// TwinCAT 3 PLC project PLC
// Title: TcError
// Company: Roald87
// Author: Roald Ruiter
// ProjectVersion: 0.2.2.0
// Description: Translate TwinCAT error codes
// ProgramVersion: 3.1.4023.0
// libraries:
//   Tc2_Standard, * (Beckhoff Automation GmbH)
//   Tc2_System, * (Beckhoff Automation GmbH)
//   Tc3_Module, * (Beckhoff Automation GmbH)
//   TcUnit,1.2.0.0,www.tcunit.org
// project tree:
//   ADS/ AdsErrorCodeDescription.TcPOU, AdsErrorCodes.TcDUT, ToAdsErrorCode.TcPOU
//   NC/ NcErrorCodes.TcDUT, ToNcErrorCode.TcPOU, NcErrorCodeDescription.TcPOU
//   NC_Tests/ ToNcErrorCode_Tests.TcPOU, NcErrorCodeDesciption_Tests.TcPOU
//   / PlcTask.TcTTO, UnitTests.TcPOU
//   Win32/ ToWin32ErrorCode.TcPOU, Win32ErrorCodeDescription.TcPOU, Win32ErrorCodes.TcDUT
//   Win32_Tests/ ToWin32ErrorCode_Tests.TcPOU, Win32ErrorCodeDesciption_Tests.TcPOU
// real-time tasks:
//   TASK PlcTask: cycle T#10ms, priority 20, ADS port 350

CONFIGURATION PLC
    RESOURCE PLC ON TwinCAT3
        TASK PlcTask(INTERVAL := T#10ms, PRIORITY := 20);
        PROGRAM UnitTests WITH PlcTask : UnitTests;
    END_RESOURCE
END_CONFIGURATION

// ---- ADS/AdsErrorCodes.TcDUT
{attribute 'qualified_only'}
{attribute 'strict'}
{attribute 'to_string'}
(*
All ADS error codes.

## Source
https://infosys.beckhoff.com/english.php?content=../content/1033/tf6701_tc3_iot_communication_mqtt/374277003.html&id=
*)
TYPE AdsErrorCodes : (
    ERR_NOERROR := 0,
    ERR_INTERNAL,
    ERR_NORTIME,
    ERR_ALLOCLOCKEDMEM,
    ERR_INSERTMAILBOX,
    ERR_WRONGRECEIVEHMSG,
    ERR_TARGETPORTNOTFOUND,
    ERR_TARGETMACHINENOTFOUND,
    ERR_UNKNOWNCMDID,
    ERR_BADTASKID,
    ERR_NOIO,
    ERR_UNKNOWNAMSCMD,
    ERR_WIN32ERROR,
    ERR_PORTNOTCONNECTED,
    ERR_INVALIDAMSLENGTH,
    ERR_INVALIDAMSNETID,
    ERR_LOWINSTLEVEL,
    ERR_NODEBUGINTAVAILABLE,
    ERR_PORTDISABLED,
    ERR_PORTALREADYCONNECTED,
    ERR_AMSSYNC_W32ERROR,
    ERR_AMSSYNC_TIMEOUT,
    ERR_AMSSYNC_AMSERROR,
    ERR_AMSSYNC_NOINDEXINMAP,
    ERR_INVALIDAMSPORT,
    ERR_NOMEMORY,
    ERR_TCPSEND,
    ERR_HOSTUNREACHABLE,
    ERR_INVALIDAMSFRAGMENT,
    ERR_TLSSEND,
    ERR_ACCESSDENIED,
    ROUTERERR_NOLOCKEDMEMORY := 1280,
    ROUTERERR_RESIZEMEMORY := 1281,
    ROUTERERR_MAILBOXFULL := 1282,
    ROUTERERR_DEBUGBOXFULL := 1283,
    ROUTERERR_UNKNOWNPORTTYPE := 1284,
    ROUTERERR_NOTINITIALIZED := 1285,
    ROUTERERR_PORTALREADYINUSE := 1286,
    ROUTERERR_NOTREGISTERED := 1287,
    ROUTERERR_NOMOREQUEUES := 1288,
    ROUTERERR_INVALIDPORT := 1289,
    ROUTERERR_NOTACTIVATED := 1290,
    ROUTERERR_FRAGMENTBOXFULL := 1291,
    ROUTERERR_FRAGMENTTIMEOUT := 1292,
    ROUTERERR_TOBEREMOVED := 1293,
    ADSERR_DEVICE_ERROR := 1792,
    ADSERR_DEVICE_SRVNOTSUPP := 1793,
    ADSERR_DEVICE_INVALIDGRP := 1794,
    ADSERR_DEVICE_INVALIDOFFSET := 1795,
    ADSERR_DEVICE_INVALIDACCESS := 1796,
    ADSERR_DEVICE_INVALIDSIZE := 1797,
    ADSERR_DEVICE_INVALIDDATA := 1798,
    ADSERR_DEVICE_NOTREADY := 1799,
    ADSERR_DEVICE_BUSY := 1800,
    ADSERR_DEVICE_INVALIDCONTEXT := 1801,
    ADSERR_DEVICE_NOMEMORY := 1802,
    ADSERR_DEVICE_INVALIDPARM := 1803,
    ADSERR_DEVICE_NOTFOUND := 1804,
    ADSERR_DEVICE_SYNTAX := 1805,
    ADSERR_DEVICE_INCOMPATIBLE := 1806,
    ADSERR_DEVICE_EXISTS := 1807,
    ADSERR_DEVICE_SYMBOLNOTFOUND := 1808,
    ADSERR_DEVICE_SYMBOLVERSIONINVALID := 1809,
    ADSERR_DEVICE_INVALIDSTATE := 1810,
    ADSERR_DEVICE_TRANSMODENOTSUPP := 1811,
    ADSERR_DEVICE_NOTIFYHNDINVALID := 1812,
    ADSERR_DEVICE_CLIENTUNKNOWN := 1813,
    ADSERR_DEVICE_NOMOREHDLS := 1814,
    ADSERR_DEVICE_INVALIDWATCHSIZE := 1815,
    ADSERR_DEVICE_NOTINIT := 1816,
    ADSERR_DEVICE_TIMEOUT := 1817,
    ADSERR_DEVICE_NOINTERFACE := 1818,
    ADSERR_DEVICE_INVALIDINTERFACE := 1819,
    ADSERR_DEVICE_INVALIDCLSID := 1820,
    ADSERR_DEVICE_INVALIDOBJID := 1821,
    ADSERR_DEVICE_PENDING := 1822,
    ADSERR_DEVICE_ABORTED := 1823,
    ADSERR_DEVICE_WARNING := 1824,
    ADSERR_DEVICE_INVALIDARRAYIDX := 1825,
    ADSERR_DEVICE_SYMBOLNOTACTIVE := 1826,
    ADSERR_DEVICE_ACCESSDENIED := 1827,
    ADSERR_DEVICE_LICENSENOTFOUND := 1828,
    ADSERR_DEVICE_LICENSEEXPIRED := 1829,
    ADSERR_DEVICE_LICENSEEXCEEDED := 1830,
    ADSERR_DEVICE_LICENSEINVALID := 1831,
    ADSERR_DEVICE_LICENSESYSTEMID := 1832,
    ADSERR_DEVICE_LICENSENOTIMELIMIT := 1833,
    ADSERR_DEVICE_LICENSEFUTUREISSUE := 1834,
    ADSERR_DEVICE_LICENSETIMETOLONG := 1835,
    ADSERR_DEVICE_EXCEPTION := 1836,
    ADSERR_DEVICE_LICENSEDUPLICATED := 1837,
    ADSERR_DEVICE_SIGNATUREINVALID := 1838,
    ADSERR_DEVICE_CERTIFICATEINVALID := 1839,
    ADSERR_DEVICE_LICENSEOEMNOTFOUND := 1840,
    ADSERR_DEVICE_LICENSERESTRICTED := 1841,
    ADSERR_DEVICE_LICENSEDEMODENIED := 1842,
    ADSERR_DEVICE_INVALIDFNCID := 1843,
    ADSERR_DEVICE_OUTOFRANGE := 1844,
    ADSERR_DEVICE_INVALIDALIGNMENT := 1845,
    ADSERR_DEVICE_LICENSEPLATFORM := 1846,
    ADSERR_DEVICE_FORWARD_PL := 1847,
    ADSERR_DEVICE_FORWARD_DL := 1848,
    ADSERR_DEVICE_FORWARD_RT := 1849,
    ADSERR_CLIENT_ERROR := 1856,
    ADSERR_CLIENT_INVALIDPARM := 1857,
    ADSERR_CLIENT_LISTEMPTY := 1858,
    ADSERR_CLIENT_VARUSED := 1859,
    ADSERR_CLIENT_DUPLINVOKEID := 1860,
    ADSERR_CLIENT_SYNCTIMEOUT := 1861,
    ADSERR_CLIENT_W32ERROR := 1862,
    ADSERR_CLIENT_TIMEOUTINVALID := 1863,
    ADSERR_CLIENT_PORTNOTOPEN := 1864,
    ADSERR_CLIENT_NOAMSADDR := 1865,
    ADSERR_CLIENT_SYNCINTERNAL := 1872,
    ADSERR_CLIENT_ADDHASH := 1873,
    ADSERR_CLIENT_REMOVEHASH := 1874,
    ADSERR_CLIENT_NOMORESYM := 1875,
    ADSERR_CLIENT_SYNCRESINVALID := 1876,
    ADSERR_CLIENT_SYNCPORTLOCKED := 1877,
    RTERR_INTERNAL := 4096,
    RTERR_BADTIMERPERIODS := 4097,
    RTERR_INVALIDTASKPTR := 4098,
    RTERR_INVALIDSTACKPTR := 4099,
    RTERR_PRIOEXISTS := 4100,
    RTERR_NOMORETCB := 4101,
    RTERR_NOMORESEMAS := 4102,
    RTERR_NOMOREQUEUES := 4103,
    RTERR_EXTIRQALREADYDEF := 4109,
    RTERR_EXTIRQNOTDEF := 4110,
    RTERR_EXTIRQINSTALLFAILED := 4111,
    RTERR_IRQLNOTLESSOREQUAL := 4112,
    RTERR_VMXNOTSUPPORTED := 4119,
    RTERR_VMXDISABLED := 4120,
    RTERR_VMXCONTROLSMISSING := 4121,
    RTERR_VMXENABLEFAILS := 4122,
    WSAETIMEDOUT := 10060,
    WSAECONNREFUSED := 10061,
    WSAEHOSTUNREACH := 10065,
    ERR_UNKNOWN := 4294967294
) UDINT;
END_TYPE

// ---- NC/NcErrorCodes.TcDUT
{attribute 'qualified_only'}
{attribute 'strict'}
(*
Some NC Error codes

Source: https://infosys.beckhoff.com/content/1033/tc3ncerrcode/1521556875.html?id=2911757239699425890
*)
TYPE NcErrorCodes : (
    NO_ERROR := 0,
    CONTROLLER_ERROR_CONTROLLER_ID_NOT_ALLOWED := 17664,
    CONTROLLER_ERROR_CONTROLLER_TYPE_NOT_ALLOWED := 17665,
    CONTROLLER_ERROR_OPERATION_MODE_CONTROLLER_NOT_ALLOWED := 17666,
    CONTROLLER_ERROR_WEIGHTING_OF_THE_VELOCITY_PRE_CONTROL_NOT_ALLOWED := 17667,
    CONTROLLER_ERROR_LAG_ERROR_MONITOR_POSITION_NOT_ALLOWED := 17668,
    CONTROLLER_ERROR_LAG_MONITORING_VELOCITY_NOT_ALLOWED := 17669,
    CONTROLLER_ERROR_LAG_ERROR_WINDOW_POSITION_NOT_ALLOWED := 17670,
    CONTROLLER_ERROR_LAG_ERROR_FILTER_TIME_POSITION_NOT_ALLOWED := 17671,
    CONTROLLER_ERROR_LAG_ERROR_WINDOW_VELOCITY_NOT_ALLOWED := 17672,
    CONTROLLER_ERROR_LAG_ERROR_FILTER_TIME_VELOCITY_NOT_ALLOWED := 17673,
    CONTROLLER_ERROR_CONTROLLER_OUTPUT_LIMITATION_OUTPUT_LIMITATION_NOT_ALLOWED := 17674,
    CONTROLLER_ERROR_PROPORTIONAL_GAIN_KV_OR_KP_CONTROLLER_NOT_ALLOWED := 17680,
    CONTROLLER_ERROR_INTEGRAL_ACTION_TIME_TN_CONTROLLER_NOT_ALLOWED_POSITION := 17681,
    CONTROLLER_ERROR_RATE_TIME_TV_CONTROLLER_NOT_ALLOWED_POSITION := 17682,
    CONTROLLER_ERROR_DAMPING_TIME_TD_CONTROLLER_NOT_ALLOWED_POSITION := 17683,
    CONTROLLER_ERROR_ACTIVATION_OF_THE_AUTOMATIC_OFFSET_CALIBRATION_NOT_ALLOWED := 17684,
    CONTROLLER_ERROR_ADDITIONAL_PROPORTIONAL_GAIN_KV_OR_KP_CONTROLLER_NOT_ALLOWED := 17685,
    CONTROLLER_ERROR_REFERENCE_VELOCITY_FOR_ADDITIONAL_PROP_GAIN_CONTROLLER_NOT_ALLOWED := 17686,
    CONTROLLER_ERROR_PROPORTIONAL_GAIN_PA_PROPORTION_NOT_ALLOWED := 17687,
    CONTROLLER_ERROR_PROPORTIONAL_GAIN_KV_CONTROLLER_NOT_ALLOWED := 17688,
    CONTROLLER_ERROR_INTEGRAL_ACTION_TIME_TN_CONTROLLER_NOT_ALLOWED_VELOCITY := 17689,
    CONTROLLER_ERROR_VELOCITY_FILTER_TIME_NOT_ALLOWED := 17692,
    CONTROLLER_ERROR_DEAD_RANGE_NOT_ALLOWED := 17693,
    CONTROLLER_ERROR_PROPORTIONAL_GAIN_KCP_NOT_ALLOWED := 17695,
    CONTROLLER_ERROR_RATE_TIME_TV_CONTROLLER_NOT_ALLOWED := 17696,
    CONTROLLER_ERROR_DAMPING_TIME_TD_CONTROLLER_NOT_ALLOWED := 17697,
    CONTROLLER_ERROR_LIMITATION_OF_THE_I_PART_NOT_ALLOWED := 17698,
    CONTROLLER_ERROR_LIMITATION_OF_THE_D_PART_NOT_ALLOWED := 17699,
    CONTROLLER_ERROR_PARAMETER_DEACTIVATION_OF_THE_I_PART_DURING_TRAVEL_NOT_ALLOWED := 17700,
    CONTROLLER_ERROR_PARAMETER_FILTER_TIME_FOR_P_T2_FILTER_NOT_ALLOWED := 17701,
    CONTROLLER_ERROR_VELOCITY_OBSERVER_PARAMETERIZED_MODE_IS_NOT_ALLOWED := 17702,
    CONTROLLER_ERROR_VELOCITY_OBSERVER_MOTOR_TORQUE_CONSTANT_KT_OR_KF_IS_NOT_ALLOWED := 17703,
    CONTROLLER_ERROR_VELOCITY_OBSERVER_MOTOR_MOMENT_OF_INERTIA_JM_IS_NOT_ALLOWED := 17704,
    CONTROLLER_ERROR_VELOCITY_OBSERVER_BANDWIDTH_F0_IS_NOT_ALLOWED := 17705,
    CONTROLLER_ERROR_VELOCITY_OBSERVER_CORRECTION_FACTOR_KC_IS_NOT_ALLOWED := 17706,
    CONTROLLER_ERROR_VELOCITY_OBSERVER_TIME_CONSTANT_T_FOR_1ST_ORDER_FILTER_NOT_ALLOWED := 17707,
    CONTROLLER_ERROR_VELOCITY_OBSERVER_AMPLITUDE_DAMPING_FOR_2ND_ORDER_FILTER_NOT_ALLOWED := 17708,
    CONTROLLER_ERROR_VELOCITY_OBSERVER_FREQUENCY_FOR_2ND_ORDER_FILTER_NOT_ALLOWED := 17709,
    CONTROLLER_ERROR_CONTROLLER_INITIALIZATION := 17728,
    CONTROLLER_ERROR_AXIS_ADDRESS := 17729,
    CONTROLLER_ERROR_DRIVE_ADDRESS := 17730,
    CONTROLLER_ERROR_LAG_ERROR_MONITOR_POSITION := 17744,
    CONTROLLER_ERROR_LAG_MONITORING_VELOCITY := 17745,
    CONTROLLER_ERROR_INTERNAL_ERROR_CONTROLERR_RANGE_AREA_ASIDE := 17824,
    CONTROLLER_ERROR_INTERNAL_ERROR_CONTROLERR_RANGE_AREA_BSIDE := 17825,
    CONTROLLER_ERROR_INTERNAL_ERROR_CONTROLERR_RANGE_QNENN := 17826,
    CONTROLLER_ERROR_INTERNAL_ERROR_CONTROLERR_RANGE_PNENN := 17827,
    CONTROLLER_ERROR_INTERNAL_ERROR_CONTROLERR_RANGE_AXISIDPRESP0 := 17828,
    ERR_UNKNOWN := 65535
);
END_TYPE

// ---- Win32/Win32ErrorCodes.TcDUT
{attribute 'qualified_only'}
{attribute 'strict'}
{attribute 'to_string'}
(*
All Win32 error codes.

## Source
https://infosys.beckhoff.com/content/1033/devicemanager/391166347.html?id=8711134805786442486
*)
TYPE Win32ErrorCodes : (
    ERROR_SUCCESS := 0,
    ERROR_INVALID_FUNCTION := 1,
    ERROR_FILE_NOT_FOUND := 2,
    ERROR_PATH_NOT_FOUND := 3,
    ERROR_TOO_MANY_OPEN_FILES := 4,
    ERROR_ACCESS_DENIED := 5,
    ERROR_INVALID_HANDLE := 6,
    ERROR_ARENA_TRASHED := 7,
    ERROR_NOT_ENOUGH_MEMORY := 8,
    ERROR_INVALID_BLOCK := 9,
    ERROR_BAD_ENVIRONMENT := 10,
    ERROR_BAD_FORMAT := 11,
    ERROR_INVALID_ACCESS := 12,
    ERROR_INVALID_DATA := 13,
    ERROR_OUTOFMEMORY := 14,
    ERROR_INVALID_DRIVE := 15,
    ERROR_CURRENT_DIRECTORY := 16,
    ERROR_NOT_SAME_DEVICE := 17,
    ERROR_NO_MORE_FILES := 18,
    ERROR_WRITE_PROTECT := 19,
    ERROR_BAD_UNIT := 20,
    ERROR_NOT_READY := 21,
    ERROR_BAD_COMMAND := 22,
    ERROR_CRC := 23,
    ERROR_BAD_LENGTH := 24,
    ERROR_SEEK := 25,
    ERROR_NOT_DOS_DISK := 26,
    ERROR_SECTOR_NOT_FOUND := 27,
    ERROR_OUT_OF_PAPER := 28,
    ERROR_WRITE_FAULT := 29,
    ERROR_READ_FAULT := 30,
    ERROR_GEN_FAILURE := 31,
    ERROR_SHARING_VIOLATION := 32,
    ERROR_LOCK_VIOLATION := 33,
    ERROR_WRONG_DISK := 34,
    ERROR_SHARING_BUFFER_EXCEEDED := 36,
    ERROR_HANDLE_EOF := 38,
    ERROR_HANDLE_DISK_FULL := 39,
    ERROR_NOT_SUPPORTED := 50,
    ERROR_REM_NOT_LIST := 51,
    ERROR_DUP_NAME := 52,
    ERROR_BAD_NETPATH := 53,
    ERROR_NETWORK_BUSY := 54,
    ERROR_DEV_NOT_EXIST := 55,
    ERROR_TOO_MANY_CMDS := 56,
    ERROR_ADAP_HDW_ERR := 57,
    ERROR_BAD_NET_RESP := 58,
    ERROR_UNEXP_NET_ERR := 59,
    ERROR_BAD_REM_ADAP := 60,
    ERROR_PRINTQ_FULL := 61,
    ERROR_NO_SPOOL_SPACE := 62,
    ERROR_PRINT_CANCELLED := 63,
    ERROR_NETNAME_DELETED := 64,
    ERROR_NETWORK_ACCESS_DENIED := 65,
    ERROR_BAD_DEV_TYPE := 66,
    ERROR_BAD_NET_NAME := 67,
    ERROR_TOO_MANY_NAMES := 68,
    ERROR_TOO_MANY_SESS := 69,
    ERROR_SHARING_PAUSED := 70,
    ERROR_REQ_NOT_ACCEP := 71,
    ERROR_REDIR_PAUSED := 72,
    ERROR_FILE_EXISTS := 80,
    ERROR_CANNOT_MAKE := 82,
    ERROR_FAIL_I24 := 83,
    ERROR_OUT_OF_STRUCTURES := 84,
    ERROR_ALREADY_ASSIGNED := 85,
    ERROR_INVALID_PASSWORD := 86,
    ERROR_INVALID_PARAMETER := 87,
    ERROR_NET_WRITE_FAULT := 88,
    ERROR_NO_PROC_SLOTS := 89,
    ERROR_TOO_MANY_SEMAPHORES := 100,
    ERROR_EXCL_SEM_ALREADY_OWNED := 101,
    ERROR_SEM_IS_SET := 102,
    ERROR_TOO_MANY_SEM_REQUESTS := 103,
    ERROR_INVALID_AT_INTERRUPT_TIME := 104,
    ERROR_SEM_OWNER_DIED := 105,
    ERROR_SEM_USER_LIMIT := 106,
    ERROR_DISK_CHANGE := 107,
    ERROR_DRIVE_LOCKED := 108,
    ERROR_BROKEN_PIPE := 109,
    ERROR_OPEN_FAILED := 110,
    ERROR_BUFFER_OVERFLOW := 111,
    ERROR_DISK_FULL := 112,
    ERROR_NO_MORE_SEARCH_HANDLES := 113,
    ERROR_INVALID_TARGET_HANDLE := 114,
    ERROR_INVALID_CATEGORY := 117,
    ERROR_INVALID_VERIFY_SWITCH := 118,
    ERROR_BAD_DRIVER_LEVEL := 119,
    ERROR_CALL_NOT_IMPLEMENTED := 120,
    ERROR_SEM_TIMEOUT := 121,
    ERROR_INSUFFICIENT_BUFFER := 122,
    ERROR_INVALID_NAME := 123,
    ERROR_INVALID_LEVEL := 124,
    ERROR_NO_VOLUME_LABEL := 125,
    ERROR_MOD_NOT_FOUND := 126,
    ERROR_PROC_NOT_FOUND := 127,
    ERROR_WAIT_NO_CHILDREN := 128,
    ERROR_CHILD_NOT_COMPLETE := 129,
    ERROR_DIRECT_ACCESS_HANDLE := 130,
    ERROR_NEGATIVE_SEEK := 131,
    ERROR_SEEK_ON_DEVICE := 132,
    ERROR_IS_JOIN_TARGET := 133,
    ERROR_IS_JOINED := 134,
    ERROR_IS_SUBSTED := 135,
    ERROR_NOT_JOINED := 136,
    ERROR_NOT_SUBSTED := 137,
    ERROR_JOIN_TO_JOIN := 138,
    ERROR_SUBST_TO_SUBST := 139,
    ERROR_JOIN_TO_SUBST := 140,
    ERROR_SUBST_TO_JOIN := 141,
    ERROR_BUSY_DRIVE := 142,
    ERROR_SAME_DRIVE := 143,
    ERROR_DIR_NOT_ROOT := 144,
    ERROR_DIR_NOT_EMPTY := 145,
    ERROR_IS_SUBST_PATH := 146,
    ERROR_IS_JOIN_PATH := 147,
    ERROR_PATH_BUSY := 148,
    ERROR_IS_SUBST_TARGET := 149,
    ERROR_SYSTEM_TRACE := 150,
    ERROR_INVALID_EVENT_COUNT := 151,
    ERROR_TOO_MANY_MUXWAITERS := 152,
    ERROR_INVALID_LIST_FORMAT := 153,
    ERROR_LABEL_TOO_LONG := 154,
    ERROR_TOO_MANY_TCBS := 155,
    ERROR_SIGNAL_REFUSED := 156,
    ERROR_DISCARDED := 157,
    ERROR_NOT_LOCKED := 158,
    ERROR_BAD_THREADID_ADDR := 159,
    ERROR_BAD_ARGUMENTS := 160,
    ERROR_BAD_PATHNAME := 161,
    ERROR_SIGNAL_PENDING := 162,
    ERROR_MAX_THRDS_REACHED := 164,
    ERROR_LOCK_FAILED := 167,
    ERROR_BUSY := 170,
    ERROR_CANCEL_VIOLATION := 173,
    ERROR_ATOMIC_LOCKS_NOT_SUPPORTED := 174,
    ERROR_INVALID_SEGMENT_NUMBER := 180,
    ERROR_INVALID_ORDINAL := 182,
    ERROR_ALREADY_EXISTS := 183,
    ERROR_INVALID_FLAG_NUMBER := 186,
    ERROR_SEM_NOT_FOUND := 187,
    ERROR_INVALID_STARTING_CODESEG := 188,
    ERROR_INVALID_STACKSEG := 189,
    ERROR_INVALID_MODULETYPE := 190,
    ERROR_INVALID_EXE_SIGNATURE := 191,
    ERROR_EXE_MARKED_INVALID := 192,
    ERROR_BAD_EXE_FORMAT := 193,
    ERROR_ITERATED_DATA_EXCEEDS_64k := 194,
    ERROR_INVALID_MINALLOCSIZE := 195,
    ERROR_DYNLINK_FROM_INVALID_RING := 196,
    ERROR_IOPL_NOT_ENABLED := 197,
    ERROR_INVALID_SEGDPL := 198,
    ERROR_AUTODATASEG_EXCEEDS_64k := 199,
    ERROR_RING2SEG_MUST_BE_MOVABLE := 200,
    ERROR_RELOC_CHAIN_XEEDS_SEGLIM := 201,
    ERROR_INFLOOP_IN_RELOC_CHAIN := 202,
    ERROR_ENVVAR_NOT_FOUND := 203,
    ERROR_NO_SIGNAL_SENT := 205,
    ERROR_FILENAME_EXCED_RANGE := 206,
    ERROR_RING2_STACK_IN_USE := 207,
    ERROR_META_EXPANSION_TOO_LONG := 208,
    ERROR_INVALID_SIGNAL_NUMBER := 209,
    ERROR_THREAD_1_INACTIVE := 210,
    ERROR_LOCKED := 212,
    ERROR_TOO_MANY_MODULES := 214,
    ERROR_NESTING_NOT_ALLOWED := 215,
    ERROR_EXE_MACHINE_TYPE_MISMATCH := 216,
    ERROR_BAD_PIPE := 230,
    ERROR_PIPE_BUSY := 231,
    ERROR_NO_DATA := 232,
    ERROR_PIPE_NOT_CONNECTED := 233,
    ERROR_MORE_DATA := 234,
    ERROR_VC_DISCONNECTED := 240,
    ERROR_INVALID_EA_NAME := 254,
    ERROR_EA_LIST_INCONSISTENT := 255,
    WAIT_TIMEOUT := 258,
    ERROR_NO_MORE_ITEMS := 259,
    ERROR_CANNOT_COPY := 266,
    ERROR_DIRECTORY := 267,
    ERROR_EAS_DIDNT_FIT := 275,
    ERROR_EA_FILE_CORRUPT := 276,
    ERROR_EA_TABLE_FULL := 277,
    ERROR_INVALID_EA_HANDLE := 278,
    ERROR_EAS_NOT_SUPPORTED := 282,
    ERROR_NOT_OWNER := 288,
    ERROR_TOO_MANY_POSTS := 298,
    ERROR_PARTIAL_COPY := 299,
    ERROR_OPLOCK_NOT_GRANTED := 300,
    ERROR_INVALID_OPLOCK_PROTOCOL := 301,
    ERROR_DISK_TOO_FRAGMENTED := 302,
    ERROR_DELETE_PENDING := 303,
    ERROR_MR_MID_NOT_FOUND := 317,
    ERROR_INVALID_ADDRESS := 487,
    ERROR_ARITHMETIC_OVERFLOW := 534,
    ERROR_PIPE_CONNECTED := 535,
    ERROR_PIPE_LISTENING := 536,
    ERROR_EA_ACCESS_DENIED := 994,
    ERROR_OPERATION_ABORTED := 995,
    ERROR_IO_INCOMPLETE := 996,
    ERROR_IO_PENDING := 997,
    ERROR_NOACCESS := 998,
    ERROR_SWAPERROR := 999,
    ERROR_STACK_OVERFLOW := 1001,
    ERROR_INVALID_MESSAGE := 1002,
    ERROR_CAN_NOT_COMPLETE := 1003,
    ERROR_INVALID_FLAGS := 1004,
    ERROR_UNRECOGNIZED_VOLUME := 1005,
    ERROR_FILE_INVALID := 1006,
    ERROR_FULLSCREEN_MODE := 1007,
    ERROR_NO_TOKEN := 1008,
    ERROR_BADDB := 1009,
    ERROR_BADKEY := 1010,
    ERROR_CANTOPEN := 1011,
    ERROR_CANTREAD := 1012,
    ERROR_CANTWRITE := 1013,
    ERROR_REGISTRY_RECOVERED := 1014,
    ERROR_REGISTRY_CORRUPT := 1015,
    ERROR_REGISTRY_IO_FAILED := 1016,
    ERROR_NOT_REGISTRY_FILE := 1017,
    ERROR_KEY_DELETED := 1018,
    ERROR_NO_LOG_SPACE := 1019,
    ERROR_KEY_HAS_CHILDREN := 1020,
    ERROR_CHILD_MUST_BE_VOLATILE := 1021,
    ERROR_NOTIFY_ENUM_DIR := 1022,
    ERROR_DEPENDENT_SERVICES_RUNNING := 1051,
    ERROR_INVALID_SERVICE_CONTROL := 1052,
    ERROR_SERVICE_REQUEST_TIMEOUT := 1053,
    ERROR_SERVICE_NO_THREAD := 1054,
    ERROR_SERVICE_DATABASE_LOCKED := 1055,
    ERROR_SERVICE_ALREADY_RUNNING := 1056,
    ERROR_INVALID_SERVICE_ACCOUNT := 1057,
    ERROR_SERVICE_DISABLED := 1058,
    ERROR_CIRCULAR_DEPENDENCY := 1059,
    ERROR_SERVICE_DOES_NOT_EXIST := 1060,
    ERROR_SERVICE_CANNOT_ACCEPT_CTRL := 1061,
    ERROR_SERVICE_NOT_ACTIVE := 1062,
    ERROR_FAILED_SERVICE_CONTROLLER_CONNECT := 1063,
    ERROR_EXCEPTION_IN_SERVICE := 1064,
    ERROR_DATABASE_DOES_NOT_EXIST := 1065,
    ERROR_SERVICE_SPECIFIC_ERROR := 1066,
    ERROR_PROCESS_ABORTED := 1067,
    ERROR_SERVICE_DEPENDENCY_FAIL := 1068,
    ERROR_SERVICE_LOGON_FAILED := 1069,
    ERROR_SERVICE_START_HANG := 1070,
    ERROR_INVALID_SERVICE_LOCK := 1071,
    ERROR_SERVICE_MARKED_FOR_DELETE := 1072,
    ERROR_SERVICE_EXISTS := 1073,
    ERROR_ALREADY_RUNNING_LKG := 1074,
    ERROR_SERVICE_DEPENDENCY_DELETED := 1075,
    ERROR_BOOT_ALREADY_ACCEPTED := 1076,
    ERROR_SERVICE_NEVER_STARTED := 1077,
    ERROR_DUPLICATE_SERVICE_NAME := 1078,
    ERROR_DIFFERENT_SERVICE_ACCOUNT := 1079,
    ERROR_CANNOT_DETECT_DRIVER_FAILURE := 1080,
    ERROR_CANNOT_DETECT_PROCESS_ABORT := 1081,
    ERROR_NO_RECOVERY_PROGRAM := 1082,
    ERROR_SERVICE_NOT_IN_EXE := 1083,
    ERROR_NOT_SAFEBOOT_SERVICE := 1084,
    ERROR_END_OF_MEDIA := 1100,
    ERROR_FILEMARK_DETECTED := 1101,
    ERROR_BEGINNING_OF_MEDIA := 1102,
    ERROR_SETMARK_DETECTED := 1103,
    ERROR_NO_DATA_DETECTED := 1104,
    ERROR_PARTITION_FAILURE := 1105,
    ERROR_INVALID_BLOCK_LENGTH := 1106,
    ERROR_DEVICE_NOT_PARTITIONED := 1107,
    ERROR_UNABLE_TO_LOCK_MEDIA := 1108,
    ERROR_UNABLE_TO_UNLOAD_MEDIA := 1109,
    ERROR_MEDIA_CHANGED := 1110,
    ERROR_BUS_RESET := 1111,
    ERROR_NO_MEDIA_IN_DRIVE := 1112,
    ERROR_NO_UNICODE_TRANSLATION := 1113,
    ERROR_DLL_INIT_FAILED := 1114,
    ERROR_SHUTDOWN_IN_PROGRESS := 1115,
    ERROR_NO_SHUTDOWN_IN_PROGRESS := 1116,
    ERROR_IO_DEVICE := 1117,
    ERROR_SERIAL_NO_DEVICE := 1118,
    ERROR_IRQ_BUSY := 1119,
    ERROR_MORE_WRITES := 1120,
    ERROR_COUNTER_TIMEOUT := 1121,
    ERROR_FLOPPY_ID_MARK_NOT_FOUND := 1122,
    ERROR_FLOPPY_WRONG_CYLINDER := 1123,
    ERROR_FLOPPY_UNKNOWN_ERROR := 1124,
    ERROR_FLOPPY_BAD_REGISTERS := 1125,
    ERROR_DISK_RECALIBRATE_FAILED := 1126,
    ERROR_DISK_OPERATION_FAILED := 1127,
    ERROR_DISK_RESET_FAILED := 1128,
    ERROR_EOM_OVERFLOW := 1129,
    ERROR_NOT_ENOUGH_SERVER_MEMORY := 1130,
    ERROR_POSSIBLE_DEADLOCK := 1131,
    ERROR_MAPPED_ALIGNMENT := 1132,
    ERROR_SET_POWER_STATE_VETOED := 1140,
    ERROR_SET_POWER_STATE_FAILED := 1141,
    ERROR_TOO_MANY_LINKS := 1142,
    ERROR_OLD_WIN_VERSION := 1150,
    ERROR_APP_WRONG_OS := 1151,
    ERROR_SINGLE_INSTANCE_APP := 1152,
    ERROR_RMODE_APP := 1153,
    ERROR_INVALID_DLL := 1154,
    ERROR_NO_ASSOCIATION := 1155,
    ERROR_DDE_FAIL := 1156,
    ERROR_DLL_NOT_FOUND := 1157,
    ERROR_NO_MORE_USER_HANDLES := 1158,
    ERROR_MESSAGE_SYNC_ONLY := 1159,
    ERROR_SOURCE_ELEMENT_EMPTY := 1160,
    ERROR_DESTINATION_ELEMENT_FULL := 1161,
    ERROR_ILLEGAL_ELEMENT_ADDRESS := 1162,
    ERROR_MAGAZINE_NOT_PRESENT := 1163,
    ERROR_DEVICE_REINITIALIZATION_NEEDED := 1164,
    ERROR_DEVICE_REQUIRES_CLEANING := 1165,
    ERROR_DEVICE_DOOR_OPEN := 1166,
    ERROR_DEVICE_NOT_CONNECTED := 1167,
    ERROR_NOT_FOUND := 1168,
    ERROR_NO_MATCH := 1169,
    ERROR_SET_NOT_FOUND := 1170,
    ERROR_POINT_NOT_FOUND := 1171,
    ERROR_NO_TRACKING_SERVICE := 1172,
    ERROR_NO_VOLUME_ID := 1173,
    ERROR_UNABLE_TO_REMOVE_REPLACED := 1175,
    ERROR_UNABLE_TO_MOVE_REPLACEMENT := 1176,
    ERROR_UNABLE_TO_MOVE_REPLACEMENT_2 := 1177,
    ERROR_JOURNAL_DELETE_IN_PROGRESS := 1178,
    ERROR_JOURNAL_NOT_ACTIVE := 1179,
    ERROR_POTENTIAL_FILE_FOUND := 1180,
    ERROR_JOURNAL_ENTRY_DELETED := 1181,
    ERROR_BAD_DEVICE := 1200,
    ERROR_CONNECTION_UNAVAIL := 1201,
    ERROR_DEVICE_ALREADY_REMEMBERED := 1202,
    ERROR_NO_NET_OR_BAD_PATH := 1203,
    ERROR_BAD_PROVIDER := 1204,
    ERROR_CANNOT_OPEN_PROFILE := 1205,
    ERROR_BAD_PROFILE := 1206,
    ERROR_NOT_CONTAINER := 1207,
    ERROR_EXTENDED_ERROR := 1208,
    ERROR_INVALID_GROUPNAME := 1209,
    ERROR_INVALID_COMPUTERNAME := 1210,
    ERROR_INVALID_EVENTNAME := 1211,
    ERROR_INVALID_DOMAINNAME := 1212,
    ERROR_INVALID_SERVICENAME := 1213,
    ERROR_INVALID_NETNAME := 1214,
    ERROR_INVALID_SHARENAME := 1215,
    ERROR_INVALID_PASSWORDNAME := 1216,
    ERROR_INVALID_MESSAGENAME := 1217,
    ERROR_INVALID_MESSAGEDEST := 1218,
    ERROR_SESSION_CREDENTIAL_CONFLICT := 1219,
    ERROR_REMOTE_SESSION_LIMIT_EXCEEDED := 1220,
    ERROR_DUP_DOMAINNAME := 1221,
    ERROR_NO_NETWORK := 1222,
    ERROR_CANCELLED := 1223,
    ERROR_USER_MAPPED_FILE := 1224,
    ERROR_CONNECTION_REFUSED := 1225,
    ERROR_GRACEFUL_DISCONNECT := 1226,
    ERROR_ADDRESS_ALREADY_ASSOCIATED := 1227,
    ERROR_ADDRESS_NOT_ASSOCIATED := 1228,
    ERROR_CONNECTION_INVALID := 1229,
    ERROR_CONNECTION_ACTIVE := 1230,
    ERROR_NETWORK_UNREACHABLE := 1231,
    ERROR_HOST_UNREACHABLE := 1232,
    ERROR_PROTOCOL_UNREACHABLE := 1233,
    ERROR_PORT_UNREACHABLE := 1234,
    ERROR_REQUEST_ABORTED := 1235,
    ERROR_CONNECTION_ABORTED := 1236,
    ERROR_RETRY := 1237,
    ERROR_CONNECTION_COUNT_LIMIT := 1238,
    ERROR_LOGIN_TIME_RESTRICTION := 1239,
    ERROR_LOGIN_WKSTA_RESTRICTION := 1240,
    ERROR_INCORRECT_ADDRESS := 1241,
    ERROR_ALREADY_REGISTERED := 1242,
    ERROR_SERVICE_NOT_FOUND := 1243,
    ERROR_NOT_AUTHENTICATED := 1244,
    ERROR_NOT_LOGGED_ON := 1245,
    ERROR_CONTINUE := 1246,
    ERROR_ALREADY_INITIALIZED := 1247,
    ERROR_NO_MORE_DEVICES := 1248,
    ERROR_NO_SUCH_SITE := 1249,
    ERROR_DOMAIN_CONTROLLER_EXISTS := 1250,
    ERROR_ONLY_IF_CONNECTED := 1251,
    ERROR_OVERRIDE_NOCHANGES := 1252,
    ERROR_BAD_USER_PROFILE := 1253,
    ERROR_NOT_SUPPORTED_ON_SBS := 1254,
    ERROR_SERVER_SHUTDOWN_IN_PROGRESS := 1255,
    ERROR_HOST_DOWN := 1256,
    ERROR_NON_ACCOUNT_SID := 1257,
    ERROR_NON_DOMAIN_SID := 1258,
    ERROR_APPHELP_BLOCK := 1259,
    ERROR_ACCESS_DISABLED_BY_POLICY := 1260,
    ERROR_REG_NAT_CONSUMPTION := 1261,
    ERROR_CSCSHARE_OFFLINE := 1262,
    ERROR_NOT_ALL_ASSIGNED := 1300,
    ERROR_SOME_NOT_MAPPED := 1301,
    ERROR_NO_QUOTAS_FOR_ACCOUNT := 1302,
    ERROR_LOCAL_USER_SESSION_KEY := 1303,
    ERROR_NULL_LM_PASSWORD := 1304,
    ERROR_UNKNOWN_REVISION := 1305,
    ERROR_REVISION_MISMATCH := 1306,
    ERROR_INVALID_OWNER := 1307,
    ERROR_INVALID_PRIMARY_GROUP := 1308,
    ERROR_NO_IMPERSONATION_TOKEN := 1309,
    ERROR_CANT_DISABLE_MANDATORY := 1310,
    ERROR_NO_LOGON_SERVERS := 1311,
    ERROR_NO_SUCH_LOGON_SESSION := 1312,
    ERROR_NO_SUCH_PRIVILEGE := 1313,
    ERROR_PRIVILEGE_NOT_HELD := 1314,
    ERROR_INVALID_ACCOUNT_NAME := 1315,
    ERROR_USER_EXISTS := 1316,
    ERROR_NO_SUCH_USER := 1317,
    ERROR_GROUP_EXISTS := 1318,
    ERROR_NO_SUCH_GROUP := 1319,
    ERROR_MEMBER_IN_GROUP := 1320,
    ERROR_MEMBER_NOT_IN_GROUP := 1321,
    ERROR_LAST_ADMIN := 1322,
    ERROR_WRONG_PASSWORD := 1323,
    ERROR_ILL_FORMED_PASSWORD := 1324,
    ERROR_PASSWORD_RESTRICTION := 1325,
    ERROR_LOGON_FAILURE := 1326,
    ERROR_ACCOUNT_RESTRICTION := 1327,
    ERROR_INVALID_LOGON_HOURS := 1328,
    ERROR_INVALID_WORKSTATION := 1329,
    ERROR_PASSWORD_EXPIRED := 1330,
    ERROR_ACCOUNT_DISABLED := 1331,
    ERROR_NONE_MAPPED := 1332,
    ERROR_TOO_MANY_LUIDS_REQUESTED := 1333,
    ERROR_LUIDS_EXHAUSTED := 1334,
    ERROR_INVALID_SUB_AUTHORITY := 1335,
    ERROR_INVALID_ACL := 1336,
    ERROR_INVALID_SID := 1337,
    ERROR_INVALID_SECURITY_DESCR := 1338,
    ERROR_BAD_INHERITANCE_ACL := 1340,
    ERROR_SERVER_DISABLED := 1341,
    ERROR_SERVER_NOT_DISABLED := 1342,
    ERROR_INVALID_ID_AUTHORITY := 1343,
    ERROR_ALLOTTED_SPACE_EXCEEDED := 1344,
    ERROR_INVALID_GROUP_ATTRIBUTES := 1345,
    ERROR_BAD_IMPERSONATION_LEVEL := 1346,
    ERROR_CANT_OPEN_ANONYMOUS := 1347,
    ERROR_BAD_VALIDATION_CLASS := 1348,
    ERROR_BAD_TOKEN_TYPE := 1349,
    ERROR_NO_SECURITY_ON_OBJECT := 1350,
    ERROR_CANT_ACCESS_DOMAIN_INFO := 1351,
    ERROR_INVALID_SERVER_STATE := 1352,
    ERROR_INVALID_DOMAIN_STATE := 1353,
    ERROR_INVALID_DOMAIN_ROLE := 1354,
    ERROR_NO_SUCH_DOMAIN := 1355,
    ERROR_DOMAIN_EXISTS := 1356,
    ERROR_DOMAIN_LIMIT_EXCEEDED := 1357,
    ERROR_INTERNAL_DB_CORRUPTION := 1358,
    ERROR_INTERNAL_ERROR := 1359,
    ERROR_GENERIC_NOT_MAPPED := 1360,
    ERROR_BAD_DESCRIPTOR_FORMAT := 1361,
    ERROR_NOT_LOGON_PROCESS := 1362,
    ERROR_LOGON_SESSION_EXISTS := 1363,
    ERROR_NO_SUCH_PACKAGE := 1364,
    ERROR_BAD_LOGON_SESSION_STATE := 1365,
    ERROR_LOGON_SESSION_COLLISION := 1366,
    ERROR_INVALID_LOGON_TYPE := 1367,
    ERROR_CANNOT_IMPERSONATE := 1368,
    ERROR_RXACT_INVALID_STATE := 1369,
    ERROR_RXACT_COMMIT_FAILURE := 1370,
    ERROR_SPECIAL_ACCOUNT := 1371,
    ERROR_SPECIAL_GROUP := 1372,
    ERROR_SPECIAL_USER := 1373,
    ERROR_MEMBERS_PRIMARY_GROUP := 1374,
    ERROR_TOKEN_ALREADY_IN_USE := 1375,
    ERROR_NO_SUCH_ALIAS := 1376,
    ERROR_MEMBER_NOT_IN_ALIAS := 1377,
    ERROR_MEMBER_IN_ALIAS := 1378,
    ERROR_ALIAS_EXISTS := 1379,
    ERROR_LOGON_NOT_GRANTED := 1380,
    ERROR_TOO_MANY_SECRETS := 1381,
    ERROR_SECRET_TOO_LONG := 1382,
    ERROR_INTERNAL_DB_ERROR := 1383,
    ERROR_TOO_MANY_CONTEXT_IDS := 1384,
    ERROR_LOGON_TYPE_NOT_GRANTED := 1385,
    ERROR_NT_CROSS_ENCRYPTION_REQUIRED := 1386,
    ERROR_NO_SUCH_MEMBER := 1387,
    ERROR_INVALID_MEMBER := 1388,
    ERROR_TOO_MANY_SIDS := 1389,
    ERROR_LM_CROSS_ENCRYPTION_REQUIRED := 1390,
    ERROR_NO_INHERITANCE := 1391,
    ERROR_FILE_CORRUPT := 1392,
    ERROR_DISK_CORRUPT := 1393,
    ERROR_NO_USER_SESSION_KEY := 1394,
    ERROR_LICENSE_QUOTA_EXCEEDED := 1395,
    ERROR_WRONG_TARGET_NAME := 1396,
    ERROR_MUTUAL_AUTH_FAILED := 1397,
    ERROR_TIME_SKEW := 1398,
    ERROR_CURRENT_DOMAIN_NOT_ALLOWED := 1399,
    ERROR_INVALID_WINDOW_HANDLE := 1400,
    ERROR_INVALID_MENU_HANDLE := 1401,
    ERROR_INVALID_CURSOR_HANDLE := 1402,
    ERROR_INVALID_ACCEL_HANDLE := 1403,
    ERROR_INVALID_HOOK_HANDLE := 1404,
    ERROR_INVALID_DWP_HANDLE := 1405,
    ERROR_TLW_WITH_WSCHILD := 1406,
    ERROR_CANNOT_FIND_WND_CLASS := 1407,
    ERROR_WINDOW_OF_OTHER_THREAD := 1408,
    ERROR_HOTKEY_ALREADY_REGISTERED := 1409,
    ERROR_CLASS_ALREADY_EXISTS := 1410,
    ERROR_CLASS_DOES_NOT_EXIST := 1411,
    ERROR_CLASS_HAS_WINDOWS := 1412,
    ERROR_INVALID_INDEX := 1413,
    ERROR_INVALID_ICON_HANDLE := 1414,
    ERROR_PRIVATE_DIALOG_INDEX := 1415,
    ERROR_LISTBOX_ID_NOT_FOUND := 1416,
    ERROR_NO_WILDCARD_CHARACTERS := 1417,
    ERROR_CLIPBOARD_NOT_OPEN := 1418,
    ERROR_HOTKEY_NOT_REGISTERED := 1419,
    ERROR_WINDOW_NOT_DIALOG := 1420,
    ERROR_CONTROL_ID_NOT_FOUND := 1421,
    ERROR_INVALID_COMBOBOX_MESSAGE := 1422,
    ERROR_WINDOW_NOT_COMBOBOX := 1423,
    ERROR_INVALID_EDIT_HEIGHT := 1424,
    ERROR_DC_NOT_FOUND := 1425,
    ERROR_INVALID_HOOK_FILTER := 1426,
    ERROR_INVALID_FILTER_PROC := 1427,
    ERROR_HOOK_NEEDS_HMOD := 1428,
    ERROR_GLOBAL_ONLY_HOOK := 1429,
    ERROR_JOURNAL_HOOK_SET := 1430,
    ERROR_HOOK_NOT_INSTALLED := 1431,
    ERROR_INVALID_LB_MESSAGE := 1432,
    ERROR_SETCOUNT_ON_BAD_LB := 1433,
    ERROR_LB_WITHOUT_TABSTOPS := 1434,
    ERROR_DESTROY_OBJECT_OF_OTHER_THREAD := 1435,
    ERROR_CHILD_WINDOW_MENU := 1436,
    ERROR_NO_SYSTEM_MENU := 1437,
    ERROR_INVALID_MSGBOX_STYLE := 1438,
    ERROR_INVALID_SPI_VALUE := 1439,
    ERROR_SCREEN_ALREADY_LOCKED := 1440,
    ERROR_HWNDS_HAVE_DIFF_PARENT := 1441,
    ERROR_NOT_CHILD_WINDOW := 1442,
    ERROR_INVALID_GW_COMMAND := 1443,
    ERROR_INVALID_THREAD_ID := 1444,
    ERROR_NON_MDICHILD_WINDOW := 1445,
    ERROR_POPUP_ALREADY_ACTIVE := 1446,
    ERROR_NO_SCROLLBARS := 1447,
    ERROR_INVALID_SCROLLBAR_RANGE := 1448,
    ERROR_INVALID_SHOWWIN_COMMAND := 1449,
    ERROR_NO_SYSTEM_RESOURCES := 1450,
    ERROR_NONPAGED_SYSTEM_RESOURCES := 1451,
    ERROR_PAGED_SYSTEM_RESOURCES := 1452,
    ERROR_WORKING_SET_QUOTA := 1453,
    ERROR_PAGEFILE_QUOTA := 1454,
    ERROR_COMMITMENT_LIMIT := 1455,
    ERROR_MENU_ITEM_NOT_FOUND := 1456,
    ERROR_INVALID_KEYBOARD_HANDLE := 1457,
    ERROR_HOOK_TYPE_NOT_ALLOWED := 1458,
    ERROR_REQUIRES_INTERACTIVE_WINDOWSTATION := 1459,
    ERROR_TIMEOUT := 1460,
    ERROR_INVALID_MONITOR_HANDLE := 1461,
    ERROR_EVENTLOG_FILE_CORRUPT := 1500,
    ERROR_EVENTLOG_CANT_START := 1501,
    ERROR_LOG_FILE_FULL := 1502,
    ERROR_EVENTLOG_FILE_CHANGED := 1503,
    ERROR_INSTALL_SERVICE_FAILURE := 1601,
    ERROR_INSTALL_USEREXIT := 1602,
    ERROR_INSTALL_FAILURE := 1603,
    ERROR_INSTALL_SUSPEND := 1604,
    ERROR_UNKNOWN_PRODUCT := 1605,
    ERROR_UNKNOWN_FEATURE := 1606,
    ERROR_UNKNOWN_COMPONENT := 1607,
    ERROR_UNKNOWN_PROPERTY := 1608,
    ERROR_INVALID_HANDLE_STATE := 1609,
    ERROR_BAD_CONFIGURATION := 1610,
    ERROR_INDEX_ABSENT := 1611,
    ERROR_INSTALL_SOURCE_ABSENT := 1612,
    ERROR_INSTALL_PACKAGE_VERSION := 1613,
    ERROR_PRODUCT_UNINSTALLED := 1614,
    ERROR_BAD_QUERY_SYNTAX := 1615,
    ERROR_INVALID_FIELD := 1616,
    ERROR_DEVICE_REMOVED := 1617,
    ERROR_INSTALL_ALREADY_RUNNING := 1618,
    ERROR_INSTALL_PACKAGE_OPEN_FAILED := 1619,
    ERROR_INSTALL_PACKAGE_INVALID := 1620,
    ERROR_INSTALL_UI_FAILURE := 1621,
    ERROR_INSTALL_LOG_FAILURE := 1622,
    ERROR_INSTALL_LANGUAGE_UNSUPPORTED := 1623,
    ERROR_INSTALL_TRANSFORM_FAILURE := 1624,
    ERROR_INSTALL_PACKAGE_REJECTED := 1625,
    ERROR_FUNCTION_NOT_CALLED := 1626,
    ERROR_FUNCTION_FAILED := 1627,
    ERROR_INVALID_TABLE := 1628,
    ERROR_DATATYPE_MISMATCH := 1629,
    ERROR_UNSUPPORTED_TYPE := 1630,
    ERROR_CREATE_FAILED := 1631,
    ERROR_INSTALL_TEMP_UNWRITABLE := 1632,
    ERROR_INSTALL_PLATFORM_UNSUPPORTED := 1633,
    ERROR_INSTALL_NOTUSED := 1634,
    ERROR_PATCH_PACKAGE_OPEN_FAILED := 1635,
    ERROR_PATCH_PACKAGE_INVALID := 1636,
    ERROR_PATCH_PACKAGE_UNSUPPORTED := 1637,
    ERROR_PRODUCT_VERSION := 1638,
    ERROR_INVALID_COMMAND_LINE := 1639,
    ERROR_INSTALL_REMOTE_DISALLOWED := 1640,
    ERROR_SUCCESS_REBOOT_INITIATED := 1641,
    ERROR_PATCH_TARGET_NOT_FOUND := 1642,
    ERROR_PATCH_PACKAGE_REJECTED := 1643,
    ERROR_INSTALL_TRANSFORM_REJECTED := 1644,
    RPC_S_INVALID_STRING_BINDING := 1700,
    RPC_S_WRONG_KIND_OF_BINDING := 1701,
    RPC_S_INVALID_BINDING := 1702,
    RPC_S_PROTSEQ_NOT_SUPPORTED := 1703,
    RPC_S_INVALID_RPC_PROTSEQ := 1704,
    RPC_S_INVALID_STRING_UUID := 1705,
    RPC_S_INVALID_ENDPOINT_FORMAT := 1706,
    RPC_S_INVALID_NET_ADDR := 1707,
    RPC_S_NO_ENDPOINT_FOUND := 1708,
    RPC_S_INVALID_TIMEOUT := 1709,
    RPC_S_OBJECT_NOT_FOUND := 1710,
    RPC_S_ALREADY_REGISTERED := 1711,
    RPC_S_TYPE_ALREADY_REGISTERED := 1712,
    RPC_S_ALREADY_LISTENING := 1713,
    RPC_S_NO_PROTSEQS_REGISTERED := 1714,
    RPC_S_NOT_LISTENING := 1715,
    RPC_S_UNKNOWN_MGR_TYPE := 1716,
    RPC_S_UNKNOWN_IF := 1717,
    RPC_S_NO_BINDINGS := 1718,
    RPC_S_NO_PROTSEQS := 1719,
    RPC_S_CANT_CREATE_ENDPOINT := 1720,
    RPC_S_OUT_OF_RESOURCES := 1721,
    RPC_S_SERVER_UNAVAILABLE := 1722,
    RPC_S_SERVER_TOO_BUSY := 1723,
    RPC_S_INVALID_NETWORK_OPTIONS := 1724,
    RPC_S_NO_CALL_ACTIVE := 1725,
    RPC_S_CALL_FAILED := 1726,
    RPC_S_CALL_FAILED_DNE := 1727,
    RPC_S_PROTOCOL_ERROR := 1728,
    RPC_S_UNSUPPORTED_TRANS_SYN := 1730,
    RPC_S_UNSUPPORTED_TYPE := 1732,
    RPC_S_INVALID_TAG := 1733,
    RPC_S_INVALID_BOUND := 1734,
    RPC_S_NO_ENTRY_NAME := 1735,
    RPC_S_INVALID_NAME_SYNTAX := 1736,
    RPC_S_UNSUPPORTED_NAME_SYNTAX := 1737,
    RPC_S_UUID_NO_ADDRESS := 1739,
    RPC_S_DUPLICATE_ENDPOINT := 1740,
    RPC_S_UNKNOWN_AUTHN_TYPE := 1741,
    RPC_S_MAX_CALLS_TOO_SMALL := 1742,
    RPC_S_STRING_TOO_LONG := 1743,
    RPC_S_PROTSEQ_NOT_FOUND := 1744,
    RPC_S_PROCNUM_OUT_OF_RANGE := 1745,
    RPC_S_BINDING_HAS_NO_AUTH := 1746,
    RPC_S_UNKNOWN_AUTHN_SERVICE := 1747,
    RPC_S_UNKNOWN_AUTHN_LEVEL := 1748,
    RPC_S_INVALID_AUTH_IDENTITY := 1749,
    RPC_S_UNKNOWN_AUTHZ_SERVICE := 1750,
    EPT_S_INVALID_ENTRY := 1751,
    EPT_S_CANT_PERFORM_OP := 1752,
    EPT_S_NOT_REGISTERED := 1753,
    RPC_S_NOTHING_TO_EXPORT := 1754,
    RPC_S_INCOMPLETE_NAME := 1755,
    RPC_S_INVALID_VERS_OPTION := 1756,
    RPC_S_NO_MORE_MEMBERS := 1757,
    RPC_S_NOT_ALL_OBJS_UNEXPORTED := 1758,
    RPC_S_INTERFACE_NOT_FOUND := 1759,
    RPC_S_ENTRY_ALREADY_EXISTS := 1760,
    RPC_S_ENTRY_NOT_FOUND := 1761,
    RPC_S_NAME_SERVICE_UNAVAILABLE := 1762,
    RPC_S_INVALID_NAF_ID := 1763,
    RPC_S_CANNOT_SUPPORT := 1764,
    RPC_S_NO_CONTEXT_AVAILABLE := 1765,
    RPC_S_INTERNAL_ERROR := 1766,
    RPC_S_ZERO_DIVIDE := 1767,
    RPC_S_ADDRESS_ERROR := 1768,
    RPC_S_FP_DIV_ZERO := 1769,
    RPC_S_FP_UNDERFLOW := 1770,
    RPC_S_FP_OVERFLOW := 1771,
    RPC_X_NO_MORE_ENTRIES := 1772,
    RPC_X_SS_CHAR_TRANS_OPEN_FAIL := 1773,
    RPC_X_SS_CHAR_TRANS_SHORT_FILE := 1774,
    RPC_X_SS_IN_NULL_CONTEXT := 1775,
    RPC_X_SS_CONTEXT_DAMAGED := 1777,
    RPC_X_SS_HANDLES_MISMATCH := 1778,
    RPC_X_SS_CANNOT_GET_CALL_HANDLE := 1779,
    RPC_X_NULL_REF_POINTER := 1780,
    RPC_X_ENUM_VALUE_OUT_OF_RANGE := 1781,
    RPC_X_BYTE_COUNT_TOO_SMALL := 1782,
    RPC_X_BAD_STUB_DATA := 1783,
    ERROR_INVALID_USER_BUFFER := 1784,
    ERROR_UNRECOGNIZED_MEDIA := 1785,
    ERROR_NO_TRUST_LSA_SECRET := 1786,
    ERROR_NO_TRUST_SAM_ACCOUNT := 1787,
    ERROR_TRUSTED_DOMAIN_FAILURE := 1788,
    ERROR_TRUSTED_RELATIONSHIP_FAILURE := 1789,
    ERROR_TRUST_FAILURE := 1790,
    RPC_S_CALL_IN_PROGRESS := 1791,
    ERROR_NETLOGON_NOT_STARTED := 1792,
    ERROR_ACCOUNT_EXPIRED := 1793,
    ERROR_REDIRECTOR_HAS_OPEN_HANDLES := 1794,
    ERROR_PRINTER_DRIVER_ALREADY_INSTALLED := 1795,
    ERROR_UNKNOWN_PORT := 1796,
    ERROR_UNKNOWN_PRINTER_DRIVER := 1797,
    ERROR_UNKNOWN_PRINTPROCESSOR := 1798,
    ERROR_INVALID_SEPARATOR_FILE := 1799,
    ERROR_INVALID_PRIORITY := 1800,
    ERROR_INVALID_PRINTER_NAME := 1801,
    ERROR_PRINTER_ALREADY_EXISTS := 1802,
    ERROR_INVALID_PRINTER_COMMAND := 1803,
    ERROR_INVALID_DATATYPE := 1804,
    ERROR_INVALID_ENVIRONMENT := 1805,
    RPC_S_NO_MORE_BINDINGS := 1806,
    ERROR_NOLOGON_INTERDOMAIN_TRUST_ACCOUNT := 1807,
    ERROR_NOLOGON_WORKSTATION_TRUST_ACCOUNT := 1808,
    ERROR_NOLOGON_SERVER_TRUST_ACCOUNT := 1809,
    ERROR_DOMAIN_TRUST_INCONSISTENT := 1810,
    ERROR_SERVER_HAS_OPEN_HANDLES := 1811,
    ERROR_RESOURCE_DATA_NOT_FOUND := 1812,
    ERROR_RESOURCE_TYPE_NOT_FOUND := 1813,
    ERROR_RESOURCE_NAME_NOT_FOUND := 1814,
    ERROR_RESOURCE_LANG_NOT_FOUND := 1815,
    ERROR_NOT_ENOUGH_QUOTA := 1816,
    RPC_S_NO_INTERFACES := 1817,
    RPC_S_CALL_CANCELLED := 1818,
    RPC_S_BINDING_INCOMPLETE := 1819,
    RPC_S_COMM_FAILURE := 1820,
    RPC_S_UNSUPPORTED_AUTHN_LEVEL := 1821,
    RPC_S_NO_PRINC_NAME := 1822,
    RPC_S_NOT_RPC_ERROR := 1823,
    RPC_S_UUID_LOCAL_ONLY := 1824,
    RPC_S_SEC_PKG_ERROR := 1825,
    RPC_S_NOT_CANCELLED := 1826,
    RPC_X_INVALID_ES_ACTION := 1827,
    RPC_X_WRONG_ES_VERSION := 1828,
    RPC_X_WRONG_STUB_VERSION := 1829,
    RPC_X_INVALID_PIPE_OBJECT := 1830,
    RPC_X_WRONG_PIPE_ORDER := 1831,
    RPC_X_WRONG_PIPE_VERSION := 1832,
    RPC_S_GROUP_MEMBER_NOT_FOUND := 1898,
    EPT_S_CANT_CREATE := 1899,
    RPC_S_INVALID_OBJECT := 1900,
    ERROR_INVALID_TIME := 1901,
    ERROR_INVALID_FORM_NAME := 1902,
    ERROR_INVALID_FORM_SIZE := 1903,
    ERROR_ALREADY_WAITING := 1904,
    ERROR_PRINTER_DELETED := 1905,
    ERROR_INVALID_PRINTER_STATE := 1906,
    ERROR_PASSWORD_MUST_CHANGE := 1907,
    ERROR_DOMAIN_CONTROLLER_NOT_FOUND := 1908,
    ERROR_ACCOUNT_LOCKED_OUT := 1909,
    OR_INVALID_OXID := 1910,
    OR_INVALID_OID := 1911,
    OR_INVALID_SET := 1912,
    RPC_S_SEND_INCOMPLETE := 1913,
    RPC_S_INVALID_ASYNC_HANDLE := 1914,
    RPC_S_INVALID_ASYNC_CALL := 1915,
    RPC_X_PIPE_CLOSED := 1916,
    RPC_X_PIPE_DISCIPLINE_ERROR := 1917,
    RPC_X_PIPE_EMPTY := 1918,
    ERROR_NO_SITENAME := 1919,
    ERROR_CANT_ACCESS_FILE := 1920,
    ERROR_CANT_RESOLVE_FILENAME := 1921,
    RPC_S_ENTRY_TYPE_MISMATCH := 1922,
    RPC_S_NOT_ALL_OBJS_EXPORTED := 1923,
    RPC_S_INTERFACE_NOT_EXPORTED := 1924,
    RPC_S_PROFILE_NOT_ADDED := 1925,
    RPC_S_PRF_ELT_NOT_ADDED := 1926,
    RPC_S_PRF_ELT_NOT_REMOVED := 1927,
    RPC_S_GRP_ELT_NOT_ADDED := 1928,
    RPC_S_GRP_ELT_NOT_REMOVED := 1929,
    ERROR_KM_DRIVER_BLOCKED := 1930,
    ERROR_INVALID_PIXEL_FORMAT := 2000,
    ERROR_BAD_DRIVER := 2001,
    ERROR_INVALID_WINDOW_STYLE := 2002,
    ERROR_METAFILE_NOT_SUPPORTED := 2003,
    ERROR_TRANSFORM_NOT_SUPPORTED := 2004,
    ERROR_CLIPPING_NOT_SUPPORTED := 2005,
    ERROR_INVALID_CMM := 2010,
    ERROR_INVALID_PROFILE := 2011,
    ERROR_TAG_NOT_FOUND := 2012,
    ERROR_TAG_NOT_PRESENT := 2013,
    ERROR_DUPLICATE_TAG := 2014,
    ERROR_PROFILE_NOT_ASSOCIATED_WITH_DEVICE := 2015,
    ERROR_PROFILE_NOT_FOUND := 2016,
    ERROR_INVALID_COLORSPACE := 2017,
    ERROR_ICM_NOT_ENABLED := 2018,
    ERROR_DELETING_ICM_XFORM := 2019,
    ERROR_INVALID_TRANSFORM := 2020,
    ERROR_COLORSPACE_MISMATCH := 2021,
    ERROR_INVALID_COLORINDEX := 2022,
    ERROR_CONNECTED_OTHER_PASSWORD := 2108,
    ERROR_BAD_USERNAME := 2202,
    ERROR_NOT_CONNECTED := 2250,
    ERROR_OPEN_FILES := 2401,
    ERROR_ACTIVE_CONNECTIONS := 2402,
    ERROR_DEVICE_IN_USE := 2404,
    ERROR_PKINIT_FAILURE := 2500,
    ERROR_SMARTCARD_SUBSYSTEM_FAILURE := 2501,
    ERROR_UNKNOWN_PRINT_MONITOR := 3000,
    ERROR_PRINTER_DRIVER_IN_USE := 3001,
    ERROR_SPOOL_FILE_NOT_FOUND := 3002,
    ERROR_SPL_NO_STARTDOC := 3003,
    ERROR_SPL_NO_ADDJOB := 3004,
    ERROR_PRINT_PROCESSOR_ALREADY_INSTALLED := 3005,
    ERROR_PRINT_MONITOR_ALREADY_INSTALLED := 3006,
    ERROR_INVALID_PRINT_MONITOR := 3007,
    ERROR_PRINT_MONITOR_IN_USE := 3008,
    ERROR_PRINTER_HAS_JOBS_QUEUED := 3009,
    ERROR_SUCCESS_REBOOT_REQUIRED := 3010,
    ERROR_SUCCESS_RESTART_REQUIRED := 3011,
    ERROR_PRINTER_NOT_FOUND := 3012,
    ERROR_WINS_INTERNAL := 4000,
    ERROR_CAN_NOT_DEL_LOCAL_WINS := 4001,
    ERROR_STATIC_INIT := 4002,
    ERROR_INC_BACKUP := 4003,
    ERROR_FULL_BACKUP := 4004,
    ERROR_REC_NON_EXISTENT := 4005,
    ERROR_RPL_NOT_ALLOWED := 4006,
    ERROR_DHCP_ADDRESS_CONFLICT := 4100,
    ERROR_WMI_GUID_NOT_FOUND := 4200,
    ERROR_WMI_INSTANCE_NOT_FOUND := 4201,
    ERROR_WMI_ITEMID_NOT_FOUND := 4202,
    ERROR_WMI_TRY_AGAIN := 4203,
    ERROR_WMI_DP_NOT_FOUND := 4204,
    ERROR_WMI_UNRESOLVED_INSTANCE_REF := 4205,
    ERROR_WMI_ALREADY_ENABLED := 4206,
    ERROR_WMI_GUID_DISCONNECTED := 4207,
    ERROR_WMI_SERVER_UNAVAILABLE := 4208,
    ERROR_WMI_DP_FAILED := 4209,
    ERROR_WMI_INVALID_MOF := 4210,
    ERROR_WMI_INVALID_REGINFO := 4211,
    ERROR_WMI_ALREADY_DISABLED := 4212,
    ERROR_WMI_READ_ONLY := 4213,
    ERROR_WMI_SET_FAILURE := 4214,
    ERROR_INVALID_MEDIA := 4300,
    ERROR_INVALID_LIBRARY := 4301,
    ERROR_INVALID_MEDIA_POOL := 4302,
    ERROR_DRIVE_MEDIA_MISMATCH := 4303,
    ERROR_MEDIA_OFFLINE := 4304,
    ERROR_LIBRARY_OFFLINE := 4305,
    ERROR_EMPTY := 4306,
    ERROR_NOT_EMPTY := 4307,
    ERROR_MEDIA_UNAVAILABLE := 4308,
    ERROR_RESOURCE_DISABLED := 4309,
    ERROR_INVALID_CLEANER := 4310,
    ERROR_UNABLE_TO_CLEAN := 4311,
    ERROR_OBJECT_NOT_FOUND := 4312,
    ERROR_DATABASE_FAILURE := 4313,
    ERROR_DATABASE_FULL := 4314,
    ERROR_MEDIA_INCOMPATIBLE := 4315,
    ERROR_RESOURCE_NOT_PRESENT := 4316,
    ERROR_INVALID_OPERATION := 4317,
    ERROR_MEDIA_NOT_AVAILABLE := 4318,
    ERROR_DEVICE_NOT_AVAILABLE := 4319,
    ERROR_REQUEST_REFUSED := 4320,
    ERROR_INVALID_DRIVE_OBJECT := 4321,
    ERROR_LIBRARY_FULL := 4322,
    ERROR_MEDIUM_NOT_ACCESSIBLE := 4323,
    ERROR_UNABLE_TO_LOAD_MEDIUM := 4324,
    ERROR_UNABLE_TO_INVENTORY_DRIVE := 4325,
    ERROR_UNABLE_TO_INVENTORY_SLOT := 4326,
    ERROR_UNABLE_TO_INVENTORY_TRANSPORT := 4327,
    ERROR_TRANSPORT_FULL := 4328,
    ERROR_CONTROLLING_IEPORT := 4329,
    ERROR_UNABLE_TO_EJECT_MOUNTED_MEDIA := 4330,
    ERROR_CLEANER_SLOT_SET := 4331,
    ERROR_CLEANER_SLOT_NOT_SET := 4332,
    ERROR_CLEANER_CARTRIDGE_SPENT := 4333,
    ERROR_UNEXPECTED_OMID := 4334,
    ERROR_CANT_DELETE_LAST_ITEM := 4335,
    ERROR_MESSAGE_EXCEEDS_MAX_SIZE := 4336,
    ERROR_VOLUME_CONTAINS_SYS_FILES := 4337,
    ERROR_INDIGENOUS_TYPE := 4338,
    ERROR_NO_SUPPORTING_DRIVES := 4339,
    ERROR_CLEANER_CARTRIDGE_INSTALLED := 4340,
    ERROR_FILE_OFFLINE := 4350,
    ERROR_REMOTE_STORAGE_NOT_ACTIVE := 4351,
    ERROR_REMOTE_STORAGE_MEDIA_ERROR := 4352,
    ERROR_NOT_A_REPARSE_POINT := 4390,
    ERROR_REPARSE_ATTRIBUTE_CONFLICT := 4391,
    ERROR_INVALID_REPARSE_DATA := 4392,
    ERROR_REPARSE_TAG_INVALID := 4393,
    ERROR_REPARSE_TAG_MISMATCH := 4394,
    ERROR_VOLUME_NOT_SIS_ENABLED := 4500,
    ERROR_DEPENDENT_RESOURCE_EXISTS := 5001,
    ERROR_DEPENDENCY_NOT_FOUND := 5002,
    ERROR_DEPENDENCY_ALREADY_EXISTS := 5003,
    ERROR_RESOURCE_NOT_ONLINE := 5004,
    ERROR_HOST_NODE_NOT_AVAILABLE := 5005,
    ERROR_RESOURCE_NOT_AVAILABLE := 5006,
    ERROR_RESOURCE_NOT_FOUND := 5007,
    ERROR_SHUTDOWN_CLUSTER := 5008,
    ERROR_CANT_EVICT_ACTIVE_NODE := 5009,
    ERROR_OBJECT_ALREADY_EXISTS := 5010,
    ERROR_OBJECT_IN_LIST := 5011,
    ERROR_GROUP_NOT_AVAILABLE := 5012,
    ERROR_GROUP_NOT_FOUND := 5013,
    ERROR_GROUP_NOT_ONLINE := 5014,
    ERROR_HOST_NODE_NOT_RESOURCE_OWNER := 5015,
    ERROR_HOST_NODE_NOT_GROUP_OWNER := 5016,
    ERROR_RESMON_CREATE_FAILED := 5017,
    ERROR_RESMON_ONLINE_FAILED := 5018,
    ERROR_RESOURCE_ONLINE := 5019,
    ERROR_QUORUM_RESOURCE := 5020,
    ERROR_NOT_QUORUM_CAPABLE := 5021,
    ERROR_CLUSTER_SHUTTING_DOWN := 5022,
    ERROR_INVALID_STATE := 5023,
    ERROR_RESOURCE_PROPERTIES_STORED := 5024,
    ERROR_NOT_QUORUM_CLASS := 5025,
    ERROR_CORE_RESOURCE := 5026,
    ERROR_QUORUM_RESOURCE_ONLINE_FAILED := 5027,
    ERROR_QUORUMLOG_OPEN_FAILED := 5028,
    ERROR_CLUSTERLOG_CORRUPT := 5029,
    ERROR_CLUSTERLOG_RECORD_EXCEEDS_MAXSIZE := 5030,
    ERROR_CLUSTERLOG_EXCEEDS_MAXSIZE := 5031,
    ERROR_CLUSTERLOG_CHKPOINT_NOT_FOUND := 5032,
    ERROR_CLUSTERLOG_NOT_ENOUGH_SPACE := 5033,
    ERROR_QUORUM_OWNER_ALIVE := 5034,
    ERROR_NETWORK_NOT_AVAILABLE := 5035,
    ERROR_NODE_NOT_AVAILABLE := 5036,
    ERROR_ALL_NODES_NOT_AVAILABLE := 5037,
    ERROR_RESOURCE_FAILED := 5038,
    ERROR_CLUSTER_INVALID_NODE := 5039,
    ERROR_CLUSTER_NODE_EXISTS := 5040,
    ERROR_CLUSTER_JOIN_IN_PROGRESS := 5041,
    ERROR_CLUSTER_NODE_NOT_FOUND := 5042,
    ERROR_CLUSTER_LOCAL_NODE_NOT_FOUND := 5043,
    ERROR_CLUSTER_NETWORK_EXISTS := 5044,
    ERROR_CLUSTER_NETWORK_NOT_FOUND := 5045,
    ERROR_CLUSTER_NETINTERFACE_EXISTS := 5046,
    ERROR_CLUSTER_NETINTERFACE_NOT_FOUND := 5047,
    ERROR_CLUSTER_INVALID_REQUEST := 5048,
    ERROR_CLUSTER_INVALID_NETWORK_PROVIDER := 5049,
    ERROR_CLUSTER_NODE_DOWN := 5050,
    ERROR_CLUSTER_NODE_UNREACHABLE := 5051,
    ERROR_CLUSTER_NODE_NOT_MEMBER := 5052,
    ERROR_CLUSTER_JOIN_NOT_IN_PROGRESS := 5053,
    ERROR_CLUSTER_INVALID_NETWORK := 5054,
    ERROR_CLUSTER_NODE_UP := 5056,
    ERROR_CLUSTER_IPADDR_IN_USE := 5057,
    ERROR_CLUSTER_NODE_NOT_PAUSED := 5058,
    ERROR_CLUSTER_NO_SECURITY_CONTEXT := 5059,
    ERROR_CLUSTER_NETWORK_NOT_INTERNAL := 5060,
    ERROR_CLUSTER_NODE_ALREADY_UP := 5061,
    ERROR_CLUSTER_NODE_ALREADY_DOWN := 5062,
    ERROR_CLUSTER_NETWORK_ALREADY_ONLINE := 5063,
    ERROR_CLUSTER_NETWORK_ALREADY_OFFLINE := 5064,
    ERROR_CLUSTER_NODE_ALREADY_MEMBER := 5065,
    ERROR_CLUSTER_LAST_INTERNAL_NETWORK := 5066,
    ERROR_CLUSTER_NETWORK_HAS_DEPENDENTS := 5067,
    ERROR_INVALID_OPERATION_ON_QUORUM := 5068,
    ERROR_DEPENDENCY_NOT_ALLOWED := 5069,
    ERROR_CLUSTER_NODE_PAUSED := 5070,
    ERROR_NODE_CANT_HOST_RESOURCE := 5071,
    ERROR_CLUSTER_NODE_NOT_READY := 5072,
    ERROR_CLUSTER_NODE_SHUTTING_DOWN := 5073,
    ERROR_CLUSTER_JOIN_ABORTED := 5074,
    ERROR_CLUSTER_INCOMPATIBLE_VERSIONS := 5075,
    ERROR_CLUSTER_MAXNUM_OF_RESOURCES_EXCEEDED := 5076,
    ERROR_CLUSTER_SYSTEM_CONFIG_CHANGED := 5077,
    ERROR_CLUSTER_RESOURCE_TYPE_NOT_FOUND := 5078,
    ERROR_CLUSTER_RESTYPE_NOT_SUPPORTED := 5079,
    ERROR_CLUSTER_RESNAME_NOT_FOUND := 5080,
    ERROR_CLUSTER_NO_RPC_PACKAGES_REGISTERED := 5081,
    ERROR_CLUSTER_OWNER_NOT_IN_PREFLIST := 5082,
    ERROR_CLUSTER_DATABASE_SEQMISMATCH := 5083,
    ERROR_RESMON_INVALID_STATE := 5084,
    ERROR_CLUSTER_GUM_NOT_LOCKER := 5085,
    ERROR_QUORUM_DISK_NOT_FOUND := 5086,
    ERROR_DATABASE_BACKUP_CORRUPT := 5087,
    ERROR_CLUSTER_NODE_ALREADY_HAS_DFS_ROOT := 5088,
    ERROR_RESOURCE_PROPERTY_UNCHANGEABLE := 5089,
    ERROR_CLUSTER_MEMBERSHIP_INVALID_STATE := 5890,
    ERROR_CLUSTER_QUORUMLOG_NOT_FOUND := 5891,
    ERROR_CLUSTER_MEMBERSHIP_HALT := 5892,
    ERROR_CLUSTER_INSTANCE_ID_MISMATCH := 5893,
    ERROR_CLUSTER_NETWORK_NOT_FOUND_FOR_IP := 5894,
    ERROR_CLUSTER_PROPERTY_DATA_TYPE_MISMATCH := 5895,
    ERROR_CLUSTER_EVICT_WITHOUT_CLEANUP := 5896,
    ERROR_ENCRYPTION_FAILED := 6000,
    ERROR_DECRYPTION_FAILED := 6001,
    ERROR_FILE_ENCRYPTED := 6002,
    ERROR_NO_RECOVERY_POLICY := 6003,
    ERROR_NO_EFS := 6004,
    ERROR_WRONG_EFS := 6005,
    ERROR_NO_USER_KEYS := 6006,
    ERROR_FILE_NOT_ENCRYPTED := 6007,
    ERROR_NOT_EXPORT_FORMAT := 6008,
    ERROR_FILE_READ_ONLY := 6009,
    ERROR_DIR_EFS_DISALLOWED := 6010,
    ERROR_EFS_SERVER_NOT_TRUSTED := 6011,
    ERROR_BAD_RECOVERY_POLICY := 6012,
    ERROR_EFS_ALG_BLOB_TOO_BIG := 6013,
    ERROR_VOLUME_NOT_SUPPORT_EFS := 6014,
    ERROR_NO_BROWSER_SERVERS_FOUND := 6118,
    SCHED_E_SERVICE_NOT_LOCALSYSTEM := 6200,
    ERROR_CTX_WINSTATION_NAME_INVALID := 7001,
    ERROR_CTX_INVALID_PD := 7002,
    ERROR_CTX_PD_NOT_FOUND := 7003,
    ERROR_CTX_WD_NOT_FOUND := 7004,
    ERROR_CTX_CANNOT_MAKE_EVENTLOG_ENTRY := 7005,
    ERROR_CTX_SERVICE_NAME_COLLISION := 7006,
    ERROR_CTX_CLOSE_PENDING := 7007,
    ERROR_CTX_NO_OUTBUF := 7008,
    ERROR_CTX_MODEM_INF_NOT_FOUND := 7009,
    ERROR_CTX_INVALID_MODEMNAME := 7010,
    ERROR_CTX_MODEM_RESPONSE_ERROR := 7011,
    ERROR_CTX_MODEM_RESPONSE_TIMEOUT := 7012,
    ERROR_CTX_MODEM_RESPONSE_NO_CARRIER := 7013,
    ERROR_CTX_MODEM_RESPONSE_NO_DIALTONE := 7014,
    ERROR_CTX_MODEM_RESPONSE_BUSY := 7015,
    ERROR_CTX_MODEM_RESPONSE_VOICE := 7016,
    ERROR_CTX_TD_ERROR := 7017,
    ERROR_CTX_WINSTATION_NOT_FOUND := 7022,
    ERROR_CTX_WINSTATION_ALREADY_EXISTS := 7023,
    ERROR_CTX_WINSTATION_BUSY := 7024,
    ERROR_CTX_BAD_VIDEO_MODE := 7025,
    ERROR_CTX_GRAPHICS_INVALID := 7035,
    ERROR_CTX_LOGON_DISABLED := 7037,
    ERROR_CTX_NOT_CONSOLE := 7038,
    ERROR_CTX_CLIENT_QUERY_TIMEOUT := 7040,
    ERROR_CTX_CONSOLE_DISCONNECT := 7041,
    ERROR_CTX_CONSOLE_CONNECT := 7042,
    ERROR_CTX_SHADOW_DENIED := 7044,
    ERROR_CTX_WINSTATION_ACCESS_DENIED := 7045,
    ERROR_CTX_INVALID_WD := 7049,
    ERROR_CTX_SHADOW_INVALID := 7050,
    ERROR_CTX_SHADOW_DISABLED := 7051,
    ERROR_CTX_CLIENT_LICENSE_IN_USE := 7052,
    ERROR_CTX_CLIENT_LICENSE_NOT_SET := 7053,
    ERROR_CTX_LICENSE_NOT_AVAILABLE := 7054,
    ERROR_CTX_LICENSE_CLIENT_INVALID := 7055,
    ERROR_CTX_LICENSE_EXPIRED := 7056,
    ERROR_CTX_SHADOW_NOT_RUNNING := 7057,
    FRS_ERR_INVALID_API_SEQUENCE := 8001,
    FRS_ERR_STARTING_SERVICE := 8002,
    FRS_ERR_STOPPING_SERVICE := 8003,
    FRS_ERR_INTERNAL_API := 8004,
    FRS_ERR_INTERNAL := 8005,
    FRS_ERR_SERVICE_COMM := 8006,
    FRS_ERR_INSUFFICIENT_PRIV := 8007,
    FRS_ERR_AUTHENTICATION := 8008,
    FRS_ERR_PARENT_INSUFFICIENT_PRIV := 8009,
    FRS_ERR_PARENT_AUTHENTICATION := 8010,
    FRS_ERR_CHILD_TO_PARENT_COMM := 8011,
    FRS_ERR_PARENT_TO_CHILD_COMM := 8012,
    FRS_ERR_SYSVOL_POPULATE := 8013,
    FRS_ERR_SYSVOL_POPULATE_TIMEOUT := 8014,
    FRS_ERR_SYSVOL_IS_BUSY := 8015,
    FRS_ERR_SYSVOL_DEMOTE := 8016,
    FRS_ERR_INVALID_SERVICE_PARAMETER := 8017,
    ERROR_DS_NOT_INSTALLED := 8200,
    ERROR_DS_MEMBERSHIP_EVALUATED_LOCALLY := 8201,
    ERROR_DS_NO_ATTRIBUTE_OR_VALUE := 8202,
    ERROR_DS_INVALID_ATTRIBUTE_SYNTAX := 8203,
    ERROR_DS_ATTRIBUTE_TYPE_UNDEFINED := 8204,
    ERROR_DS_ATTRIBUTE_OR_VALUE_EXISTS := 8205,
    ERROR_DS_BUSY := 8206,
    ERROR_DS_UNAVAILABLE := 8207,
    ERROR_DS_NO_RIDS_ALLOCATED := 8208,
    ERROR_DS_NO_MORE_RIDS := 8209,
    ERROR_DS_INCORRECT_ROLE_OWNER := 8210,
    ERROR_DS_RIDMGR_INIT_ERROR := 8211,
    ERROR_DS_OBJ_CLASS_VIOLATION := 8212,
    ERROR_DS_CANT_ON_NON_LEAF := 8213,
    ERROR_DS_CANT_ON_RDN := 8214,
    ERROR_DS_CANT_MOD_OBJ_CLASS := 8215,
    ERROR_DS_CROSS_DOM_MOVE_ERROR := 8216,
    ERROR_DS_GC_NOT_AVAILABLE := 8217,
    ERROR_SHARED_POLICY := 8218,
    ERROR_POLICY_OBJECT_NOT_FOUND := 8219,
    ERROR_POLICY_ONLY_IN_DS := 8220,
    ERROR_PROMOTION_ACTIVE := 8221,
    ERROR_NO_PROMOTION_ACTIVE := 8222,
    ERROR_DS_OPERATIONS_ERROR := 8224,
    ERROR_DS_PROTOCOL_ERROR := 8225,
    ERROR_DS_TIMELIMIT_EXCEEDED := 8226,
    ERROR_DS_SIZELIMIT_EXCEEDED := 8227,
    ERROR_DS_ADMIN_LIMIT_EXCEEDED := 8228,
    ERROR_DS_COMPARE_FALSE := 8229,
    ERROR_DS_COMPARE_TRUE := 8230,
    ERROR_DS_AUTH_METHOD_NOT_SUPPORTED := 8231,
    ERROR_DS_STRONG_AUTH_REQUIRED := 8232,
    ERROR_DS_INAPPROPRIATE_AUTH := 8233,
    ERROR_DS_AUTH_UNKNOWN := 8234,
    ERROR_DS_REFERRAL := 8235,
    ERROR_DS_UNAVAILABLE_CRIT_EXTENSION := 8236,
    ERROR_DS_CONFIDENTIALITY_REQUIRED := 8237,
    ERROR_DS_INAPPROPRIATE_MATCHING := 8238,
    ERROR_DS_CONSTRAINT_VIOLATION := 8239,
    ERROR_DS_NO_SUCH_OBJECT := 8240,
    ERROR_DS_ALIAS_PROBLEM := 8241,
    ERROR_DS_INVALID_DN_SYNTAX := 8242,
    ERROR_DS_IS_LEAF := 8243,
    ERROR_DS_ALIAS_DEREF_PROBLEM := 8244,
    ERROR_DS_UNWILLING_TO_PERFORM := 8245,
    ERROR_DS_LOOP_DETECT := 8246,
    ERROR_DS_NAMING_VIOLATION := 8247,
    ERROR_DS_OBJECT_RESULTS_TOO_LARGE := 8248,
    ERROR_DS_AFFECTS_MULTIPLE_DSAS := 8249,
    ERROR_DS_SERVER_DOWN := 8250,
    ERROR_DS_LOCAL_ERROR := 8251,
    ERROR_DS_ENCODING_ERROR := 8252,
    ERROR_DS_DECODING_ERROR := 8253,
    ERROR_DS_FILTER_UNKNOWN := 8254,
    ERROR_DS_PARAM_ERROR := 8255,
    ERROR_DS_NOT_SUPPORTED := 8256,
    ERROR_DS_NO_RESULTS_RETURNED := 8257,
    ERROR_DS_CONTROL_NOT_FOUND := 8258,
    ERROR_DS_CLIENT_LOOP := 8259,
    ERROR_DS_REFERRAL_LIMIT_EXCEEDED := 8260,
    ERROR_DS_SORT_CONTROL_MISSING := 8261,
    ERROR_DS_OFFSET_RANGE_ERROR := 8262,
    ERROR_DS_ROOT_MUST_BE_NC := 8301,
    ERROR_DS_ADD_REPLICA_INHIBITED := 8302,
    ERROR_DS_ATT_NOT_DEF_IN_SCHEMA := 8303,
    ERROR_DS_MAX_OBJ_SIZE_EXCEEDED := 8304,
    ERROR_DS_OBJ_STRING_NAME_EXISTS := 8305,
    ERROR_DS_NO_RDN_DEFINED_IN_SCHEMA := 8306,
    ERROR_DS_RDN_DOESNT_MATCH_SCHEMA := 8307,
    ERROR_DS_NO_REQUESTED_ATTS_FOUND := 8308,
    ERROR_DS_USER_BUFFER_TO_SMALL := 8309,
    ERROR_DS_ATT_IS_NOT_ON_OBJ := 8310,
    ERROR_DS_ILLEGAL_MOD_OPERATION := 8311,
    ERROR_DS_OBJ_TOO_LARGE := 8312,
    ERROR_DS_BAD_INSTANCE_TYPE := 8313,
    ERROR_DS_MASTERDSA_REQUIRED := 8314,
    ERROR_DS_OBJECT_CLASS_REQUIRED := 8315,
    ERROR_DS_MISSING_REQUIRED_ATT := 8316,
    ERROR_DS_ATT_NOT_DEF_FOR_CLASS := 8317,
    ERROR_DS_ATT_ALREADY_EXISTS := 8318,
    ERROR_DS_CANT_ADD_ATT_VALUES := 8320,
    ERROR_DS_SINGLE_VALUE_CONSTRAINT := 8321,
    ERROR_DS_RANGE_CONSTRAINT := 8322,
    ERROR_DS_ATT_VAL_ALREADY_EXISTS := 8323,
    ERROR_DS_CANT_REM_MISSING_ATT := 8324,
    ERROR_DS_CANT_REM_MISSING_ATT_VAL := 8325,
    ERROR_DS_ROOT_CANT_BE_SUBREF := 8326,
    ERROR_DS_NO_CHAINING := 8327,
    ERROR_DS_NO_CHAINED_EVAL := 8328,
    ERROR_DS_NO_PARENT_OBJECT := 8329,
    ERROR_DS_PARENT_IS_AN_ALIAS := 8330,
    ERROR_DS_CANT_MIX_MASTER_AND_REPS := 8331,
    ERROR_DS_CHILDREN_EXIST := 8332,
    ERROR_DS_OBJ_NOT_FOUND := 8333,
    ERROR_DS_ALIASED_OBJ_MISSING := 8334,
    ERROR_DS_BAD_NAME_SYNTAX := 8335,
    ERROR_DS_ALIAS_POINTS_TO_ALIAS := 8336,
    ERROR_DS_CANT_DEREF_ALIAS := 8337,
    ERROR_DS_OUT_OF_SCOPE := 8338,
    ERROR_DS_OBJECT_BEING_REMOVED := 8339,
    ERROR_DS_CANT_DELETE_DSA_OBJ := 8340,
    ERROR_DS_GENERIC_ERROR := 8341,
    ERROR_DS_DSA_MUST_BE_INT_MASTER := 8342,
    ERROR_DS_CLASS_NOT_DSA := 8343,
    ERROR_DS_INSUFF_ACCESS_RIGHTS := 8344,
    ERROR_DS_ILLEGAL_SUPERIOR := 8345,
    ERROR_DS_ATTRIBUTE_OWNED_BY_SAM := 8346,
    ERROR_DS_NAME_TOO_MANY_PARTS := 8347,
    ERROR_DS_NAME_TOO_LONG := 8348,
    ERROR_DS_NAME_VALUE_TOO_LONG := 8349,
    ERROR_DS_NAME_UNPARSEABLE := 8350,
    ERROR_DS_NAME_TYPE_UNKNOWN := 8351,
    ERROR_DS_NOT_AN_OBJECT := 8352,
    ERROR_DS_SEC_DESC_TOO_SHORT := 8353,
    ERROR_DS_SEC_DESC_INVALID := 8354,
    ERROR_DS_NO_DELETED_NAME := 8355,
    ERROR_DS_SUBREF_MUST_HAVE_PARENT := 8356,
    ERROR_DS_NCNAME_MUST_BE_NC := 8357,
    ERROR_DS_CANT_ADD_SYSTEM_ONLY := 8358,
    ERROR_DS_CLASS_MUST_BE_CONCRETE := 8359,
    ERROR_DS_INVALID_DMD := 8360,
    ERROR_DS_OBJ_GUID_EXISTS := 8361,
    ERROR_DS_NOT_ON_BACKLINK := 8362,
    ERROR_DS_NO_CROSSREF_FOR_NC := 8363,
    ERROR_DS_SHUTTING_DOWN := 8364,
    ERROR_DS_UNKNOWN_OPERATION := 8365,
    ERROR_DS_INVALID_ROLE_OWNER := 8366,
    ERROR_DS_COULDNT_CONTACT_FSMO := 8367,
    ERROR_DS_CROSS_NC_DN_RENAME := 8368,
    ERROR_DS_CANT_MOD_SYSTEM_ONLY := 8369,
    ERROR_DS_REPLICATOR_ONLY := 8370,
    ERROR_DS_OBJ_CLASS_NOT_DEFINED := 8371,
    ERROR_DS_OBJ_CLASS_NOT_SUBCLASS := 8372,
    ERROR_DS_NAME_REFERENCE_INVALID := 8373,
    ERROR_DS_CROSS_REF_EXISTS := 8374,
    ERROR_DS_CANT_DEL_MASTER_CROSSREF := 8375,
    ERROR_DS_SUBTREE_NOTIFY_NOT_NC_HEAD := 8376,
    ERROR_DS_NOTIFY_FILTER_TOO_COMPLEX := 8377,
    ERROR_DS_DUP_RDN := 8378,
    ERROR_DS_DUP_OID := 8379,
    ERROR_DS_DUP_MAPI_ID := 8380,
    ERROR_DS_DUP_SCHEMA_ID_GUID := 8381,
    ERROR_DS_DUP_LDAP_DISPLAY_NAME := 8382,
    ERROR_DS_SEMANTIC_ATT_TEST := 8383,
    ERROR_DS_SYNTAX_MISMATCH := 8384,
    ERROR_DS_EXISTS_IN_MUST_HAVE := 8385,
    ERROR_DS_EXISTS_IN_MAY_HAVE := 8386,
    ERROR_DS_NONEXISTENT_MAY_HAVE := 8387,
    ERROR_DS_NONEXISTENT_MUST_HAVE := 8388,
    ERROR_DS_AUX_CLS_TEST_FAIL := 8389,
    ERROR_DS_NONEXISTENT_POSS_SUP := 8390,
    ERROR_DS_SUB_CLS_TEST_FAIL := 8391,
    ERROR_DS_BAD_RDN_ATT_ID_SYNTAX := 8392,
    ERROR_DS_EXISTS_IN_AUX_CLS := 8393,
    ERROR_DS_EXISTS_IN_SUB_CLS := 8394,
    ERROR_DS_EXISTS_IN_POSS_SUP := 8395,
    ERROR_DS_RECALCSCHEMA_FAILED := 8396,
    ERROR_DS_TREE_DELETE_NOT_FINISHED := 8397,
    ERROR_DS_CANT_DELETE := 8398,
    ERROR_DS_ATT_SCHEMA_REQ_ID := 8399,
    ERROR_DS_BAD_ATT_SCHEMA_SYNTAX := 8400,
    ERROR_DS_CANT_CACHE_ATT := 8401,
    ERROR_DS_CANT_CACHE_CLASS := 8402,
    ERROR_DS_CANT_REMOVE_ATT_CACHE := 8403,
    ERROR_DS_CANT_REMOVE_CLASS_CACHE := 8404,
    ERROR_DS_CANT_RETRIEVE_DN := 8405,
    ERROR_DS_MISSING_SUPREF := 8406,
    ERROR_DS_CANT_RETRIEVE_INSTANCE := 8407,
    ERROR_DS_CODE_INCONSISTENCY := 8408,
    ERROR_DS_DATABASE_ERROR := 8409,
    ERROR_DS_GOVERNSID_MISSING := 8410,
    ERROR_DS_MISSING_EXPECTED_ATT := 8411,
    ERROR_DS_NCNAME_MISSING_CR_REF := 8412,
    ERROR_DS_SECURITY_CHECKING_ERROR := 8413,
    ERROR_DS_SCHEMA_NOT_LOADED := 8414,
    ERROR_DS_SCHEMA_ALLOC_FAILED := 8415,
    ERROR_DS_ATT_SCHEMA_REQ_SYNTAX := 8416,
    ERROR_DS_GCVERIFY_ERROR := 8417,
    ERROR_DS_DRA_SCHEMA_MISMATCH := 8418,
    ERROR_DS_CANT_FIND_DSA_OBJ := 8419,
    ERROR_DS_CANT_FIND_EXPECTED_NC := 8420,
    ERROR_DS_CANT_FIND_NC_IN_CACHE := 8421,
    ERROR_DS_CANT_RETRIEVE_CHILD := 8422,
    ERROR_DS_SECURITY_ILLEGAL_MODIFY := 8423,
    ERROR_DS_CANT_REPLACE_HIDDEN_REC := 8424,
    ERROR_DS_BAD_HIERARCHY_FILE := 8425,
    ERROR_DS_BUILD_HIERARCHY_TABLE_FAILED := 8426,
    ERROR_DS_CONFIG_PARAM_MISSING := 8427,
    ERROR_DS_COUNTING_AB_INDICES_FAILED := 8428,
    ERROR_DS_HIERARCHY_TABLE_MALLOC_FAILED := 8429,
    ERROR_DS_INTERNAL_FAILURE := 8430,
    ERROR_DS_UNKNOWN_ERROR := 8431,
    ERROR_DS_ROOT_REQUIRES_CLASS_TOP := 8432,
    ERROR_DS_REFUSING_FSMO_ROLES := 8433,
    ERROR_DS_MISSING_FSMO_SETTINGS := 8434,
    ERROR_DS_UNABLE_TO_SURRENDER_ROLES := 8435,
    ERROR_DS_DRA_GENERIC := 8436,
    ERROR_DS_DRA_INVALID_PARAMETER := 8437,
    ERROR_DS_DRA_BUSY := 8438,
    ERROR_DS_DRA_BAD_DN := 8439,
    ERROR_DS_DRA_BAD_NC := 8440,
    ERROR_DS_DRA_DN_EXISTS := 8441,
    ERROR_DS_DRA_INTERNAL_ERROR := 8442,
    ERROR_DS_DRA_INCONSISTENT_DIT := 8443,
    ERROR_DS_DRA_CONNECTION_FAILED := 8444,
    ERROR_DS_DRA_BAD_INSTANCE_TYPE := 8445,
    ERROR_DS_DRA_OUT_OF_MEM := 8446,
    ERROR_DS_DRA_MAIL_PROBLEM := 8447,
    ERROR_DS_DRA_REF_ALREADY_EXISTS := 8448,
    ERROR_DS_DRA_REF_NOT_FOUND := 8449,
    ERROR_DS_DRA_OBJ_IS_REP_SOURCE := 8450,
    ERROR_DS_DRA_DB_ERROR := 8451,
    ERROR_DS_DRA_NO_REPLICA := 8452,
    ERROR_DS_DRA_ACCESS_DENIED := 8453,
    ERROR_DS_DRA_NOT_SUPPORTED := 8454,
    ERROR_DS_DRA_RPC_CANCELLED := 8455,
    ERROR_DS_DRA_SOURCE_DISABLED := 8456,
    ERROR_DS_DRA_SINK_DISABLED := 8457,
    ERROR_DS_DRA_NAME_COLLISION := 8458,
    ERROR_DS_DRA_SOURCE_REINSTALLED := 8459,
    ERROR_DS_DRA_MISSING_PARENT := 8460,
    ERROR_DS_DRA_PREEMPTED := 8461,
    ERROR_DS_DRA_ABANDON_SYNC := 8462,
    ERROR_DS_DRA_SHUTDOWN := 8463,
    ERROR_DS_DRA_INCOMPATIBLE_PARTIAL_SET := 8464,
    ERROR_DS_DRA_SOURCE_IS_PARTIAL_REPLICA := 8465,
    ERROR_DS_DRA_EXTN_CONNECTION_FAILED := 8466,
    ERROR_DS_INSTALL_SCHEMA_MISMATCH := 8467,
    ERROR_DS_DUP_LINK_ID := 8468,
    ERROR_DS_NAME_ERROR_RESOLVING := 8469,
    ERROR_DS_NAME_ERROR_NOT_FOUND := 8470,
    ERROR_DS_NAME_ERROR_NOT_UNIQUE := 8471,
    ERROR_DS_NAME_ERROR_NO_MAPPING := 8472,
    ERROR_DS_NAME_ERROR_DOMAIN_ONLY := 8473,
    ERROR_DS_NAME_ERROR_NO_SYNTACTICAL_MAPPING := 8474,
    ERROR_DS_CONSTRUCTED_ATT_MOD := 8475,
    ERROR_DS_WRONG_OM_OBJ_CLASS := 8476,
    ERROR_DS_DRA_REPL_PENDING := 8477,
    ERROR_DS_DS_REQUIRED := 8478,
    ERROR_DS_INVALID_LDAP_DISPLAY_NAME := 8479,
    ERROR_DS_NON_BASE_SEARCH := 8480,
    ERROR_DS_CANT_RETRIEVE_ATTS := 8481,
    ERROR_DS_BACKLINK_WITHOUT_LINK := 8482,
    ERROR_DS_EPOCH_MISMATCH := 8483,
    ERROR_DS_SRC_NAME_MISMATCH := 8484,
    ERROR_DS_SRC_AND_DST_NC_IDENTICAL := 8485,
    ERROR_DS_DST_NC_MISMATCH := 8486,
    ERROR_DS_NOT_AUTHORITIVE_FOR_DST_NC := 8487,
    ERROR_DS_SRC_GUID_MISMATCH := 8488,
    ERROR_DS_CANT_MOVE_DELETED_OBJECT := 8489,
    ERROR_DS_PDC_OPERATION_IN_PROGRESS := 8490,
    ERROR_DS_CROSS_DOMAIN_CLEANUP_REQD := 8491,
    ERROR_DS_ILLEGAL_XDOM_MOVE_OPERATION := 8492,
    ERROR_DS_CANT_WITH_ACCT_GROUP_MEMBERSHPS := 8493,
    ERROR_DS_NC_MUST_HAVE_NC_PARENT := 8494,
    ERROR_DS_CR_IMPOSSIBLE_TO_VALIDATE := 8495,
    ERROR_DS_DST_DOMAIN_NOT_NATIVE := 8496,
    ERROR_DS_MISSING_INFRASTRUCTURE_CONTAINER := 8497,
    ERROR_DS_CANT_MOVE_ACCOUNT_GROUP := 8498,
    ERROR_DS_CANT_MOVE_RESOURCE_GROUP := 8499,
    ERROR_DS_INVALID_SEARCH_FLAG := 8500,
    ERROR_DS_NO_TREE_DELETE_ABOVE_NC := 8501,
    ERROR_DS_COULDNT_LOCK_TREE_FOR_DELETE := 8502,
    ERROR_DS_COULDNT_IDENTIFY_OBJECTS_FOR_TREE_DELETE := 8503,
    ERROR_DS_SAM_INIT_FAILURE := 8504,
    ERROR_DS_SENSITIVE_GROUP_VIOLATION := 8505,
    ERROR_DS_CANT_MOD_PRIMARYGROUPID := 8506,
    ERROR_DS_ILLEGAL_BASE_SCHEMA_MOD := 8507,
    ERROR_DS_NONSAFE_SCHEMA_CHANGE := 8508,
    ERROR_DS_SCHEMA_UPDATE_DISALLOWED := 8509,
    ERROR_DS_CANT_CREATE_UNDER_SCHEMA := 8510,
    ERROR_DS_INSTALL_NO_SRC_SCH_VERSION := 8511,
    ERROR_DS_INSTALL_NO_SCH_VERSION_IN_INIFILE := 8512,
    ERROR_DS_INVALID_GROUP_TYPE := 8513,
    ERROR_DS_NO_NEST_GLOBALGROUP_IN_MIXEDDOMAIN := 8514,
    ERROR_DS_NO_NEST_LOCALGROUP_IN_MIXEDDOMAIN := 8515,
    ERROR_DS_GLOBAL_CANT_HAVE_LOCAL_MEMBER := 8516,
    ERROR_DS_GLOBAL_CANT_HAVE_UNIVERSAL_MEMBER := 8517,
    ERROR_DS_UNIVERSAL_CANT_HAVE_LOCAL_MEMBER := 8518,
    ERROR_DS_GLOBAL_CANT_HAVE_CROSSDOMAIN_MEMBER := 8519,
    ERROR_DS_LOCAL_CANT_HAVE_CROSSDOMAIN_LOCAL_MEMBER := 8520,
    ERROR_DS_HAVE_PRIMARY_MEMBERS := 8521,
    ERROR_DS_STRING_SD_CONVERSION_FAILED := 8522,
    ERROR_DS_NAMING_MASTER_GC := 8523,
    ERROR_DS_LOOKUP_FAILURE := 8524,
    ERROR_DS_COULDNT_UPDATE_SPNS := 8525,
    ERROR_DS_CANT_RETRIEVE_SD := 8526,
    ERROR_DS_KEY_NOT_UNIQUE := 8527,
    ERROR_DS_WRONG_LINKED_ATT_SYNTAX := 8528,
    ERROR_DS_SAM_NEED_BOOTKEY_PASSWORD := 8529,
    ERROR_DS_SAM_NEED_BOOTKEY_FLOPPY := 8530,
    ERROR_DS_CANT_START := 8531,
    ERROR_DS_INIT_FAILURE := 8532,
    ERROR_DS_NO_PKT_PRIVACY_ON_CONNECTION := 8533,
    ERROR_DS_SOURCE_DOMAIN_IN_FOREST := 8534,
    ERROR_DS_DESTINATION_DOMAIN_NOT_IN_FOREST := 8535,
    ERROR_DS_DESTINATION_AUDITING_NOT_ENABLED := 8536,
    ERROR_DS_CANT_FIND_DC_FOR_SRC_DOMAIN := 8537,
    ERROR_DS_SRC_OBJ_NOT_GROUP_OR_USER := 8538,
    ERROR_DS_SRC_SID_EXISTS_IN_FOREST := 8539,
    ERROR_DS_SRC_AND_DST_OBJECT_CLASS_MISMATCH := 8540,
    ERROR_SAM_INIT_FAILURE := 8541,
    ERROR_DS_DRA_SCHEMA_INFO_SHIP := 8542,
    ERROR_DS_DRA_SCHEMA_CONFLICT := 8543,
    ERROR_DS_DRA_EARLIER_SCHEMA_CONLICT := 8544,
    ERROR_DS_DRA_OBJ_NC_MISMATCH := 8545,
    ERROR_DS_NC_STILL_HAS_DSAS := 8546,
    ERROR_DS_GC_REQUIRED := 8547,
    ERROR_DS_LOCAL_MEMBER_OF_LOCAL_ONLY := 8548,
    ERROR_DS_NO_FPO_IN_UNIVERSAL_GROUPS := 8549,
    ERROR_DS_CANT_ADD_TO_GC := 8550,
    ERROR_DS_NO_CHECKPOINT_WITH_PDC := 8551,
    ERROR_DS_SOURCE_AUDITING_NOT_ENABLED := 8552,
    ERROR_DS_CANT_CREATE_IN_NONDOMAIN_NC := 8553,
    ERROR_DS_INVALID_NAME_FOR_SPN := 8554,
    ERROR_DS_FILTER_USES_CONTRUCTED_ATTRS := 8555,
    ERROR_DS_UNICODEPWD_NOT_IN_QUOTES := 8556,
    ERROR_DS_MACHINE_ACCOUNT_QUOTA_EXCEEDED := 8557,
    ERROR_DS_MUST_BE_RUN_ON_DST_DC := 8558,
    ERROR_DS_SRC_DC_MUST_BE_SP4_OR_GREATER := 8559,
    ERROR_DS_CANT_TREE_DELETE_CRITICAL_OBJ := 8560,
    ERROR_DS_INIT_FAILURE_CONSOLE := 8561,
    ERROR_DS_SAM_INIT_FAILURE_CONSOLE := 8562,
    ERROR_DS_FOREST_VERSION_TOO_HIGH := 8563,
    ERROR_DS_DOMAIN_VERSION_TOO_HIGH := 8564,
    ERROR_DS_FOREST_VERSION_TOO_LOW := 8565,
    ERROR_DS_DOMAIN_VERSION_TOO_LOW := 8566,
    ERROR_DS_INCOMPATIBLE_VERSION := 8567,
    ERROR_DS_LOW_DSA_VERSION := 8568,
    ERROR_DS_NO_BEHAVIOR_VERSION_IN_MIXEDDOMAIN := 8569,
    ERROR_DS_NOT_SUPPORTED_SORT_ORDER := 8570,
    ERROR_DS_NAME_NOT_UNIQUE := 8571,
    ERROR_DS_MACHINE_ACCOUNT_CREATED_PRENT4 := 8572,
    ERROR_DS_OUT_OF_VERSION_STORE := 8573,
    ERROR_DS_INCOMPATIBLE_CONTROLS_USED := 8574,
    ERROR_DS_NO_REF_DOMAIN := 8575,
    ERROR_DS_RESERVED_LINK_ID := 8576,
    ERROR_DS_LINK_ID_NOT_AVAILABLE := 8577,
    ERROR_DS_AG_CANT_HAVE_UNIVERSAL_MEMBER := 8578,
    ERROR_DS_MODIFYDN_DISALLOWED_BY_INSTANCE_TYPE := 8579,
    ERROR_DS_NO_OBJECT_MOVE_IN_SCHEMA_NC := 8580,
    ERROR_DS_MODIFYDN_DISALLOWED_BY_FLAG := 8581,
    ERROR_DS_MODIFYDN_WRONG_GRANDPARENT := 8582,
    ERROR_DS_NAME_ERROR_TRUST_REFERRAL := 8583,
    ERROR_NOT_SUPPORTED_ON_STANDARD_SERVER := 8584,
    ERROR_DS_CANT_ACCESS_REMOTE_PART_OF_AD := 8585,
    ERROR_DS_CR_IMPOSSIBLE_TO_VALIDATE_V2 := 8586,
    ERROR_DS_THREAD_LIMIT_EXCEEDED := 8587,
    ERROR_DS_NOT_CLOSEST := 8588,
    DNS_ERROR_RCODE_FORMAT_ERROR := 9001,
    DNS_ERROR_RCODE_SERVER_FAILURE := 9002,
    DNS_ERROR_RCODE_NAME_ERROR := 9003,
    DNS_ERROR_RCODE_NOT_IMPLEMENTED := 9004,
    DNS_ERROR_RCODE_REFUSED := 9005,
    DNS_ERROR_RCODE_YXDOMAIN := 9006,
    DNS_ERROR_RCODE_YXRRSET := 9007,
    DNS_ERROR_RCODE_NXRRSET := 9008,
    DNS_ERROR_RCODE_NOTAUTH := 9009,
    DNS_ERROR_RCODE_NOTZONE := 9010,
    DNS_ERROR_RCODE_BADSIG := 9016,
    DNS_ERROR_RCODE_BADKEY := 9017,
    DNS_ERROR_RCODE_BADTIME := 9018,
    DNS_INFO_NO_RECORDS := 9501,
    DNS_ERROR_BAD_PACKET := 9502,
    DNS_ERROR_NO_PACKET := 9503,
    DNS_ERROR_RCODE := 9504,
    DNS_ERROR_UNSECURE_PACKET := 9505,
    DNS_ERROR_INVALID_TYPE := 9551,
    DNS_ERROR_INVALID_IP_ADDRESS := 9552,
    DNS_ERROR_INVALID_PROPERTY := 9553,
    DNS_ERROR_TRY_AGAIN_LATER := 9554,
    DNS_ERROR_NOT_UNIQUE := 9555,
    DNS_ERROR_NON_RFC_NAME := 9556,
    DNS_STATUS_FQDN := 9557,
    DNS_STATUS_DOTTED_NAME := 9558,
    DNS_STATUS_SINGLE_PART_NAME := 9559,
    DNS_ERROR_INVALID_NAME_CHAR := 9560,
    DNS_ERROR_NUMERIC_NAME := 9561,
    DNS_ERROR_ZONE_DOES_NOT_EXIST := 9601,
    DNS_ERROR_NO_ZONE_INFO := 9602,
    DNS_ERROR_INVALID_ZONE_OPERATION := 9603,
    DNS_ERROR_ZONE_CONFIGURATION_ERROR := 9604,
    DNS_ERROR_ZONE_HAS_NO_SOA_RECORD := 9605,
    DNS_ERROR_ZONE_HAS_NO_NS_RECORDS := 9606,
    DNS_ERROR_ZONE_LOCKED := 9607,
    DNS_ERROR_ZONE_CREATION_FAILED := 9608,
    DNS_ERROR_ZONE_ALREADY_EXISTS := 9609,
    DNS_ERROR_AUTOZONE_ALREADY_EXISTS := 9610,
    DNS_ERROR_INVALID_ZONE_TYPE := 9611,
    DNS_ERROR_SECONDARY_REQUIRES_MASTER_IP := 9612,
    DNS_ERROR_ZONE_NOT_SECONDARY := 9613,
    DNS_ERROR_NEED_SECONDARY_ADDRESSES := 9614,
    DNS_ERROR_WINS_INIT_FAILED := 9615,
    DNS_ERROR_NEED_WINS_SERVERS := 9616,
    DNS_ERROR_NBSTAT_INIT_FAILED := 9617,
    DNS_ERROR_SOA_DELETE_INVALID := 9618,
    DNS_ERROR_FORWARDER_ALREADY_EXISTS := 9619,
    DNS_ERROR_PRIMARY_REQUIRES_DATAFILE := 9651,
    DNS_ERROR_INVALID_DATAFILE_NAME := 9652,
    DNS_ERROR_DATAFILE_OPEN_FAILURE := 9653,
    DNS_ERROR_FILE_WRITEBACK_FAILED := 9654,
    DNS_ERROR_DATAFILE_PARSING := 9655,
    DNS_ERROR_RECORD_DOES_NOT_EXIST := 9701,
    DNS_ERROR_RECORD_FORMAT := 9702,
    DNS_ERROR_NODE_CREATION_FAILED := 9703,
    DNS_ERROR_UNKNOWN_RECORD_TYPE := 9704,
    DNS_ERROR_RECORD_TIMED_OUT := 9705,
    DNS_ERROR_NAME_NOT_IN_ZONE := 9706,
    DNS_ERROR_CNAME_LOOP := 9707,
    DNS_ERROR_NODE_IS_CNAME := 9708,
    DNS_ERROR_CNAME_COLLISION := 9709,
    DNS_ERROR_RECORD_ONLY_AT_ZONE_ROOT := 9710,
    DNS_ERROR_RECORD_ALREADY_EXISTS := 9711,
    DNS_ERROR_SECONDARY_DATA := 9712,
    DNS_ERROR_NO_CREATE_CACHE_DATA := 9713,
    DNS_ERROR_NAME_DOES_NOT_EXIST := 9714,
    DNS_WARNING_PTR_CREATE_FAILED := 9715,
    DNS_WARNING_DOMAIN_UNDELETED := 9716,
    DNS_ERROR_DS_UNAVAILABLE := 9717,
    DNS_ERROR_DS_ZONE_ALREADY_EXISTS := 9718,
    DNS_ERROR_NO_BOOTFILE_IF_DS_ZONE := 9719,
    DNS_INFO_AXFR_COMPLETE := 9751,
    DNS_ERROR_AXFR := 9752,
    DNS_INFO_ADDED_LOCAL_WINS := 9753,
    DNS_STATUS_CONTINUE_NEEDED := 9801,
    DNS_ERROR_NO_TCPIP := 9851,
    DNS_ERROR_NO_DNS_SERVERS := 9852,
    DNS_ERROR_DP_DOES_NOT_EXIST := 9901,
    DNS_ERROR_DP_ALREADY_EXISTS := 9902,
    DNS_ERROR_DP_NOT_ENLISTED := 9903,
    DNS_ERROR_DP_ALREADY_ENLISTED := 9904,
    WSAEINTR := 10004,
    WSAEBADF := 10009,
    WSAEACCES := 10013,
    WSAEFAULT := 10014,
    WSAEINVAL := 10022,
    WSAEMFILE := 10024,
    WSAEWOULDBLOCK := 10035,
    WSAEINPROGRESS := 10036,
    WSAEALREADY := 10037,
    WSAENOTSOCK := 10038,
    WSAEDESTADDRREQ := 10039,
    WSAEMSGSIZE := 10040,
    WSAEPROTOTYPE := 10041,
    WSAENOPROTOOPT := 10042,
    WSAEPROTONOSUPPORT := 10043,
    WSAESOCKTNOSUPPORT := 10044,
    WSAEOPNOTSUPP := 10045,
    WSAEPFNOSUPPORT := 10046,
    WSAEAFNOSUPPORT := 10047,
    WSAEADDRINUSE := 10048,
    WSAEADDRNOTAVAIL := 10049,
    WSAENETDOWN := 10050,
    WSAENETUNREACH := 10051,
    WSAENETRESET := 10052,
    WSAECONNABORTED := 10053,
    WSAECONNRESET := 10054,
    WSAENOBUFS := 10055,
    WSAEISCONN := 10056,
    WSAENOTCONN := 10057,
    WSAESHUTDOWN := 10058,
    WSAETOOMANYREFS := 10059,
    WSAETIMEDOUT := 10060,
    WSAECONNREFUSED := 10061,
    WSAELOOP := 10062,
    WSAENAMETOOLONG := 10063,
    WSAEHOSTDOWN := 10064,
    WSAEHOSTUNREACH := 10065,
    WSAENOTEMPTY := 10066,
    WSAEPROCLIM := 10067,
    WSAEUSERS := 10068,
    WSAEDQUOT := 10069,
    WSAESTALE := 10070,
    WSAEREMOTE := 10071,
    WSASYSNOTREADY := 10091,
    WSAVERNOTSUPPORTED := 10092,
    WSANOTINITIALISED := 10093,
    WSAEDISCON := 10101,
    WSAENOMORE := 10102,
    WSAECANCELLED := 10103,
    WSAEINVALIDPROCTABLE := 10104,
    WSAEINVALIDPROVIDER := 10105,
    WSAEPROVIDERFAILEDINIT := 10106,
    WSASYSCALLFAILURE := 10107,
    WSASERVICE_NOT_FOUND := 10108,
    WSATYPE_NOT_FOUND := 10109,
    WSA_E_NO_MORE := 10110,
    WSA_E_CANCELLED := 10111,
    WSAEREFUSED := 10112,
    WSAHOST_NOT_FOUND := 11001,
    WSATRY_AGAIN := 11002,
    WSANO_RECOVERY := 11003,
    WSANO_DATA := 11004,
    WSA_QOS_RECEIVERS := 11005,
    WSA_QOS_SENDERS := 11006,
    WSA_QOS_NO_SENDERS := 11007,
    WSA_QOS_NO_RECEIVERS := 11008,
    WSA_QOS_REQUEST_CONFIRMED := 11009,
    WSA_QOS_ADMISSION_FAILURE := 11010,
    WSA_QOS_POLICY_FAILURE := 11011,
    WSA_QOS_BAD_STYLE := 11012,
    WSA_QOS_BAD_OBJECT := 11013,
    WSA_QOS_TRAFFIC_CTRL_ERROR := 11014,
    WSA_QOS_GENERIC_ERROR := 11015,
    WSA_QOS_ESERVICETYPE := 11016,
    WSA_QOS_EFLOWSPEC := 11017,
    WSA_QOS_EPROVSPECBUF := 11018,
    WSA_QOS_EFILTERSTYLE := 11019,
    WSA_QOS_EFILTERTYPE := 11020,
    WSA_QOS_EFILTERCOUNT := 11021,
    WSA_QOS_EOBJLENGTH := 11022,
    WSA_QOS_EFLOWCOUNT := 11023,
    WSA_QOS_EUNKNOWNPSOBJ := 11024,
    WSA_QOS_EPOLICYOBJ := 11025,
    WSA_QOS_EFLOWDESC := 11026,
    WSA_QOS_EPSFLOWSPEC := 11027,
    WSA_QOS_EPSFILTERSPEC := 11028,
    WSA_QOS_ESDMODEOBJ := 11029,
    WSA_QOS_ESHAPERATEOBJ := 11030,
    WSA_QOS_RESERVED_PETYPE := 11031,
    ERROR_SXS_SECTION_NOT_FOUND := 12000,
    ERROR_SXS_CANT_GEN_ACTCTX := 12001,
    ERROR_SXS_INVALID_ACTCTXDATA_FORMAT := 12002,
    ERROR_SXS_ASSEMBLY_NOT_FOUND := 12003,
    ERROR_SXS_MANIFEST_FORMAT_ERROR := 12004,
    ERROR_SXS_MANIFEST_PARSE_ERROR := 12005,
    ERROR_SXS_ACTIVATION_CONTEXT_DISABLED := 12006,
    ERROR_SXS_KEY_NOT_FOUND := 12007,
    ERROR_SXS_VERSION_CONFLICT := 12008,
    ERROR_SXS_WRONG_SECTION_TYPE := 12009,
    ERROR_SXS_THREAD_QUERIES_DISABLED := 12010,
    ERROR_SXS_PROCESS_DEFAULT_ALREADY_SET := 12011,
    ERROR_SXS_UNKNOWN_ENCODING_GROUP := 12012,
    ERROR_SXS_UNKNOWN_ENCODING := 12013,
    ERROR_SXS_INVALID_XML_NAMESPACE_URI := 12014,
    ERROR_SXS_ROOT_MANIFEST_DEPENDENCY_NOT_INSTALLED := 12015,
    ERROR_SXS_LEAF_MANIFEST_DEPENDENCY_NOT_INSTALLED := 12016,
    ERROR_SXS_INVALID_ASSEMBLY_IDENTITY_ATTRIBUTE := 12017,
    ERROR_SXS_MANIFEST_MISSING_REQUIRED_DEFAULT_NAMESPACE := 12018,
    ERROR_SXS_MANIFEST_INVALID_REQUIRED_DEFAULT_NAMESPACE := 12019,
    ERROR_SXS_PRIVATE_MANIFEST_CROSS_PATH_WITH_REPARSE_POINT := 12020,
    ERROR_SXS_DUPLICATE_DLL_NAME := 12021,
    ERROR_SXS_DUPLICATE_WINDOWCLASS_NAME := 12022,
    ERROR_SXS_DUPLICATE_CLSID := 12023,
    ERROR_SXS_DUPLICATE_IID := 12024,
    ERROR_SXS_DUPLICATE_TLBID := 12025,
    ERROR_SXS_DUPLICATE_PROGID := 12026,
    ERROR_SXS_DUPLICATE_ASSEMBLY_NAME := 12027,
    ERROR_SXS_FILE_HASH_MISMATCH := 12028,
    ERROR_SXS_POLICY_PARSE_ERROR := 12029,
    ERROR_SXS_XML_E_MISSINGQUOTE := 12030,
    ERROR_SXS_XML_E_COMMENTSYNTAX := 12031,
    ERROR_SXS_XML_E_BADSTARTNAMECHAR := 12032,
    ERROR_SXS_XML_E_BADNAMECHAR := 12033,
    ERROR_SXS_XML_E_BADCHARINSTRING := 12034,
    ERROR_SXS_XML_E_XMLDECLSYNTAX := 12035,
    ERROR_SXS_XML_E_BADCHARDATA := 12036,
    ERROR_SXS_XML_E_MISSINGWHITESPACE := 12037,
    ERROR_SXS_XML_E_EXPECTINGTAGEND := 12038,
    ERROR_SXS_XML_E_MISSINGSEMICOLON := 12039,
    ERROR_SXS_XML_E_UNBALANCEDPAREN := 12040,
    ERROR_SXS_XML_E_INTERNALERROR := 12041,
    ERROR_SXS_XML_E_UNEXPECTED_WHITESPACE := 12042,
    ERROR_SXS_XML_E_INCOMPLETE_ENCODING := 12043,
    ERROR_SXS_XML_E_MISSING_PAREN := 12044,
    ERROR_SXS_XML_E_EXPECTINGCLOSEQUOTE := 12045,
    ERROR_SXS_XML_E_MULTIPLE_COLONS := 12046,
    ERROR_SXS_XML_E_INVALID_DECIMAL := 12047,
    ERROR_SXS_XML_E_INVALID_HEXIDECIMAL := 12048,
    ERROR_SXS_XML_E_INVALID_UNICODE := 12049,
    ERROR_SXS_XML_E_WHITESPACEORQUESTIONMARK := 12050,
    ERROR_SXS_XML_E_UNEXPECTEDENDTAG := 12051,
    ERROR_SXS_XML_E_UNCLOSEDTAG := 12052,
    ERROR_SXS_XML_E_DUPLICATEATTRIBUTE := 12053,
    ERROR_SXS_XML_E_MULTIPLEROOTS := 12054,
    ERROR_SXS_XML_E_INVALIDATROOTLEVEL := 12055,
    ERROR_SXS_XML_E_BADXMLDECL := 12056,
    ERROR_SXS_XML_E_MISSINGROOT := 12057,
    ERROR_SXS_XML_E_UNEXPECTEDEOF := 12058,
    ERROR_SXS_XML_E_BADPEREFINSUBSET := 12059,
    ERROR_SXS_XML_E_UNCLOSEDSTARTTAG := 12060,
    ERROR_SXS_XML_E_UNCLOSEDENDTAG := 12061,
    ERROR_SXS_XML_E_UNCLOSEDSTRING := 12062,
    ERROR_SXS_XML_E_UNCLOSEDCOMMENT := 12063,
    ERROR_SXS_XML_E_UNCLOSEDDECL := 12064,
    ERROR_SXS_XML_E_UNCLOSEDCDATA := 12065,
    ERROR_SXS_XML_E_RESERVEDNAMESPACE := 12066,
    ERROR_SXS_XML_E_INVALIDENCODING := 12067,
    ERROR_SXS_XML_E_INVALIDSWITCH := 12068,
    ERROR_SXS_XML_E_BADXMLCASE := 12069,
    ERROR_SXS_XML_E_INVALID_STANDALONE := 12070,
    ERROR_SXS_XML_E_UNEXPECTED_STANDALONE := 12071,
    ERROR_SXS_XML_E_INVALID_VERSION := 12072,
    ERROR_SXS_XML_E_MISSINGEQUALS := 12073,
    ERROR_IPSEC_QM_POLICY_EXISTS := 13000,
    ERROR_IPSEC_QM_POLICY_NOT_FOUND := 13001,
    ERROR_IPSEC_QM_POLICY_IN_USE := 13002,
    ERROR_IPSEC_MM_POLICY_EXISTS := 13003,
    ERROR_IPSEC_MM_POLICY_NOT_FOUND := 13004,
    ERROR_IPSEC_MM_POLICY_IN_USE := 13005,
    ERROR_IPSEC_MM_FILTER_EXISTS := 13006,
    ERROR_IPSEC_MM_FILTER_NOT_FOUND := 13007,
    ERROR_IPSEC_TRANSPORT_FILTER_EXISTS := 13008,
    ERROR_IPSEC_TRANSPORT_FILTER_NOT_FOUND := 13009,
    ERROR_IPSEC_MM_AUTH_EXISTS := 13010,
    ERROR_IPSEC_MM_AUTH_NOT_FOUND := 13011,
    ERROR_IPSEC_MM_AUTH_IN_USE := 13012,
    ERROR_IPSEC_DEFAULT_MM_POLICY_NOT_FOUND := 13013,
    ERROR_IPSEC_DEFAULT_MM_AUTH_NOT_FOUND := 13014,
    ERROR_IPSEC_DEFAULT_QM_POLICY_NOT_FOUND := 13015,
    ERROR_IPSEC_TUNNEL_FILTER_EXISTS := 13016,
    ERROR_IPSEC_TUNNEL_FILTER_NOT_FOUND := 13017,
    ERROR_IPSEC_MM_FILTER_PENDING_DELETION := 13018,
    ERROR_IPSEC_TRANSPORT_FILTER_PENDING_DELETION := 13019,
    ERROR_IPSEC_TUNNEL_FILTER_PENDING_DELETION := 13020,
    ERROR_IPSEC_MM_POLICY_PENDING_DELETION := 13021,
    ERROR_IPSEC_MM_AUTH_PENDING_DELETION := 13022,
    ERROR_IPSEC_QM_POLICY_PENDING_DELETION := 13023,
    ERROR_IPSEC_IKE_AUTH_FAIL := 13801,
    ERROR_IPSEC_IKE_ATTRIB_FAIL := 13802,
    ERROR_IPSEC_IKE_NEGOTIATION_PENDING := 13803,
    ERROR_IPSEC_IKE_GENERAL_PROCESSING_ERROR := 13804,
    ERROR_IPSEC_IKE_TIMED_OUT := 13805,
    ERROR_IPSEC_IKE_NO_CERT := 13806,
    ERROR_IPSEC_IKE_SA_DELETED := 13807,
    ERROR_IPSEC_IKE_SA_REAPED := 13808,
    ERROR_IPSEC_IKE_MM_ACQUIRE_DROP := 13809,
    ERROR_IPSEC_IKE_QM_ACQUIRE_DROP := 13810,
    ERROR_IPSEC_IKE_QUEUE_DROP_MM := 13811,
    ERROR_IPSEC_IKE_QUEUE_DROP_NO_MM := 13812,
    ERROR_IPSEC_IKE_DROP_NO_RESPONSE := 13813,
    ERROR_IPSEC_IKE_MM_DELAY_DROP := 13814,
    ERROR_IPSEC_IKE_QM_DELAY_DROP := 13815,
    ERROR_IPSEC_IKE_ERROR := 13816,
    ERROR_IPSEC_IKE_CRL_FAILED := 13817,
    ERROR_IPSEC_IKE_INVALID_KEY_USAGE := 13818,
    ERROR_IPSEC_IKE_INVALID_CERT_TYPE := 13819,
    ERROR_IPSEC_IKE_NO_PRIVATE_KEY := 13820,
    ERROR_IPSEC_IKE_DH_FAIL := 13822,
    ERROR_IPSEC_IKE_INVALID_HEADER := 13824,
    ERROR_IPSEC_IKE_NO_POLICY := 13825,
    ERROR_IPSEC_IKE_INVALID_SIGNATURE := 13826,
    ERROR_IPSEC_IKE_KERBEROS_ERROR := 13827,
    ERROR_IPSEC_IKE_NO_PUBLIC_KEY := 13828,
    ERROR_IPSEC_IKE_PROCESS_ERR := 13829,
    ERROR_IPSEC_IKE_PROCESS_ERR_SA := 13830,
    ERROR_IPSEC_IKE_PROCESS_ERR_PROP := 13831,
    ERROR_IPSEC_IKE_PROCESS_ERR_TRANS := 13832,
    ERROR_IPSEC_IKE_PROCESS_ERR_KE := 13833,
    ERROR_IPSEC_IKE_PROCESS_ERR_ID := 13834,
    ERROR_IPSEC_IKE_PROCESS_ERR_CERT := 13835,
    ERROR_IPSEC_IKE_PROCESS_ERR_CERT_REQ := 13836,
    ERROR_IPSEC_IKE_PROCESS_ERR_HASH := 13837,
    ERROR_IPSEC_IKE_PROCESS_ERR_SIG := 13838,
    ERROR_IPSEC_IKE_PROCESS_ERR_NONCE := 13839,
    ERROR_IPSEC_IKE_PROCESS_ERR_NOTIFY := 13840,
    ERROR_IPSEC_IKE_PROCESS_ERR_DELETE := 13841,
    ERROR_IPSEC_IKE_PROCESS_ERR_VENDOR := 13842,
    ERROR_IPSEC_IKE_INVALID_PAYLOAD := 13843,
    ERROR_IPSEC_IKE_LOAD_SOFT_SA := 13844,
    ERROR_IPSEC_IKE_SOFT_SA_TORN_DOWN := 13845,
    ERROR_IPSEC_IKE_INVALID_COOKIE := 13846,
    ERROR_IPSEC_IKE_NO_PEER_CERT := 13847,
    ERROR_IPSEC_IKE_PEER_CRL_FAILED := 13848,
    ERROR_IPSEC_IKE_POLICY_CHANGE := 13849,
    ERROR_IPSEC_IKE_NO_MM_POLICY := 13850,
    ERROR_IPSEC_IKE_NOTCBPRIV := 13851,
    ERROR_IPSEC_IKE_SECLOADFAIL := 13852,
    ERROR_IPSEC_IKE_FAILSSPINIT := 13853,
    ERROR_IPSEC_IKE_FAILQUERYSSP := 13854,
    ERROR_IPSEC_IKE_SRVACQFAIL := 13855,
    ERROR_IPSEC_IKE_SRVQUERYCRED := 13856,
    ERROR_IPSEC_IKE_GETSPIFAIL := 13857,
    ERROR_IPSEC_IKE_INVALID_FILTER := 13858,
    ERROR_IPSEC_IKE_OUT_OF_MEMORY := 13859,
    ERROR_IPSEC_IKE_ADD_UPDATE_KEY_FAILED := 13860,
    ERROR_IPSEC_IKE_INVALID_POLICY := 13861,
    ERROR_IPSEC_IKE_UNKNOWN_DOI := 13862,
    ERROR_IPSEC_IKE_INVALID_SITUATION := 13863,
    ERROR_IPSEC_IKE_DH_FAILURE := 13864,
    ERROR_IPSEC_IKE_INVALID_GROUP := 13865,
    ERROR_IPSEC_IKE_ENCRYPT := 13866,
    ERROR_IPSEC_IKE_DECRYPT := 13867,
    ERROR_IPSEC_IKE_POLICY_MATCH := 13868,
    ERROR_IPSEC_IKE_UNSUPPORTED_ID := 13869,
    ERROR_IPSEC_IKE_INVALID_HASH := 13870,
    ERROR_IPSEC_IKE_INVALID_HASH_ALG := 13871,
    ERROR_IPSEC_IKE_INVALID_HASH_SIZE := 13872,
    ERROR_IPSEC_IKE_INVALID_ENCRYPT_ALG := 13873,
    ERROR_IPSEC_IKE_INVALID_AUTH_ALG := 13874,
    ERROR_IPSEC_IKE_INVALID_SIG := 13875,
    ERROR_IPSEC_IKE_LOAD_FAILED := 13876,
    ERROR_IPSEC_IKE_RPC_DELETE := 13877,
    ERROR_IPSEC_IKE_BENIGN_REINIT := 13878,
    ERROR_IPSEC_IKE_INVALID_RESPONDER_LIFETIME_NOTIFY := 13879,
    ERROR_IPSEC_IKE_QM_LIMIT_REAP := 13880,
    ERROR_IPSEC_IKE_INVALID_CERT_KEYLEN := 13881,
    ERROR_IPSEC_IKE_MM_LIMIT := 13882,
    ERROR_IPSEC_IKE_NEGOTIATION_DISABLED := 13883,
    ERROR_IPSEC_IKE_QM_LIMIT := 13884,
    ERR_UNKNOWN := 4294967294
) UDINT;
END_TYPE

// ---- UnitTests.TcPOU
{attribute 'hide'}
PROGRAM UnitTests
VAR
    {attribute 'analysis' := '-33'}
    toWin32ErrorCode_Tests : ToWin32ErrorCode_Tests;
    {attribute 'analysis' := '-33'}
    win32ErrorCodeDescription_Tests : Win32ErrorCodeDesciption_Tests;
    {attribute 'analysis' := '-33'}
    toNcErrorCode_Tests : ToNcErrorCode_Tests;
    {attribute 'analysis' := '-33'}
    ncErrorCodeDescription_Tests : NcErrorCodeDesciption_Tests;
END_VAR

TcUnit.RUN();

END_PROGRAM

// ---- Win32_Tests/ToWin32ErrorCode_Tests.TcPOU
{attribute 'hide'}
FUNCTION_BLOCK ToWin32ErrorCode_Tests EXTENDS TcUnit.FB_TestSuite

ConversionOfValidErrorCode();
ConversionOfInvalidErrorCode();

METHOD ConversionOfInvalidErrorCode
TcUnit.TEST('ConversionOfInvalidErrorCode');

AssertEquals_UDINT(
    Expected:=Win32ErrorCodes.ERR_UNKNOWN,
    Actual:=ToWin32ErrorCode(1234567),
    Message:='Error conversion not correct.'
);

TcUnit.TEST_FINISHED();
END_METHOD

METHOD ConversionOfValidErrorCode
TcUnit.TEST('ConversionOfValidErrorCode');

AssertEquals_UDINT(
    Expected:=Win32ErrorCodes.ERROR_FILE_EXISTS,
    Actual:=ToWin32ErrorCode(80),
    Message:='Error conversion not correct.'
);

TcUnit.TEST_FINISHED();
END_METHOD

END_FUNCTION_BLOCK

// ---- Win32/ToWin32ErrorCode.TcPOU
(*
Convert an Win32 error code of type UDINT to the Win32ErrorCodes datatype.

## Example
```
win32ErrorId := 82;
win32ErrorCode := ToWin32ErrorCode(win32ErrorId); // ERROR_CANNOT_MAKE;
```

## Source
https://infosys.beckhoff.com/content/1033/devicemanager/391166347.html?id=8711134805786442486
*)
FUNCTION ToWin32ErrorCode : Win32ErrorCodes
VAR_INPUT
    errorCode : UDINT;
END_VAR

